KUKA KRL program: MyProgram_081().src

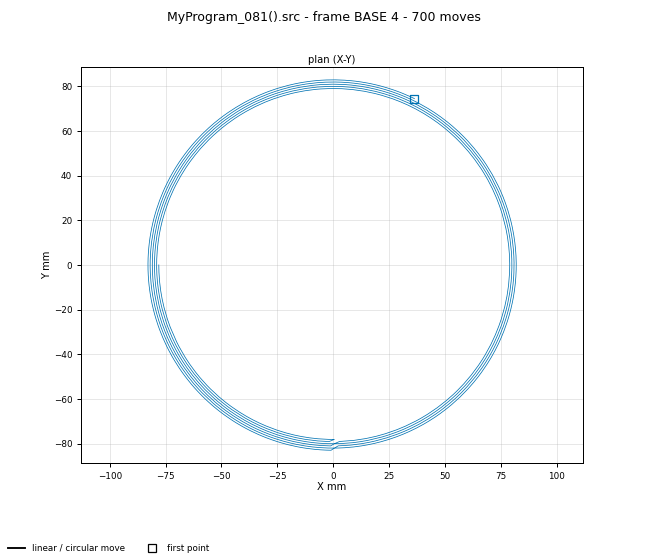
[picture p0: tool path of MyProgram_081().src in frame BASE 4, 700 of 700 moves have a stored position in this frame; points joined in program order, loops and branches not executed]
&ACCESS RVP
&REL 1
&PARAM TEMPLATE = C:\KRC\Roboter\Template\vorgabe
&PARAM EDITMASK = *
DEF MyProgram_081()
; ---- Setting reference (Base) ----
$BASE = BASE_DATA[4]

; --------------------------
; ---- Setting tool (TCP) ----
$TOOL = TOOL_DATA[3]
; --------------------------

$VEL.CP = VEL_APROX_PRINT
Startdeposition()
$VEL.CP = VEL_PRINT
LIN {X 36.3666,Y 74.5111,Z 82,A 58.7177,B 24.8945,C -2.3712,E1 25.0694,E2 385.953} C_DIS
LIN {X 34.2905,Y 75.4877,Z 82,A 60.1854,B 24.8947,C -2.3694,E1 25.0657,E2 384.4932} C_DIS
LIN {X 32.4557,Y 76.2947,Z 82,A 61.5848,B 24.8945,C -2.3714,E1 25.0621,E2 383.0926} C_DIS
LIN {X 30.7867,Y 76.9845,Z 82,A 62.9666,B 24.894,C -2.3768,E1 25.0585,E2 381.7013} C_DIS
LIN {X 28.8882,Y 77.7168,Z 82,A 64.37,B 24.8939,C -2.378,E1 25.0549,E2 380.298} C_DIS
LIN {X 26.9089,Y 78.4237,Z 82,A 65.9427,B 24.8934,C -2.3829,E1 25.0507,E2 378.7167} C_DIS
LIN {X 24.0041,Y 79.361,Z 82,A 67.8847,B 24.8938,C -2.3794,E1 25.0456,E2 376.7865} C_DIS
LIN {X 22.1137,Y 79.9088,Z 82,A 69.2831,B 24.8936,C -2.3815,E1 25.0418,E2 375.3855} C_DIS
LIN {X 19.68,Y 80.5411,Z 82,A 71.0984,B 24.8933,C -2.3849,E1 25.0369,E2 373.5648} C_DIS
LIN {X 17.1067,Y 81.1279,Z 82,A 72.799,B 24.8935,C -2.3821,E1 25.0322,E2 371.8732} C_DIS
LIN {X 15.1105,Y 81.5232,Z 82,A 74.2055,B 24.8935,C -2.3827,E1 25.0284,E2 370.4669} C_DIS
LIN {X 12.5489,Y 81.9555,Z 82,A 76.1064,B 24.8931,C -2.3864,E1 25.0231,E2 368.559} C_DIS
LIN {X 10.083,Y 82.2964,Z 82,A 77.7189,B 24.8934,C -2.3835,E1 25.0187,E2 366.9546} C_DIS
LIN {X 8.1268,Y 82.5129,Z 82,A 79.2702,B 24.8929,C -2.3894,E1 25.0143,E2 365.3903} C_DIS
LIN {X 5.0842,Y 82.7562,Z 82,A 81.2283,B 24.8933,C -2.385,E1 25.0089,E2 363.4437} C_DIS
LIN {X 2.8241,Y 82.863,Z 82,A 82.6559,B 24.8936,C -2.3809,E1 25.005,E2 362.0264} C_DIS
LIN {X 0.9507,Y 82.9063,Z 82,A 84.0039,B 24.8936,C -2.3823,E1 25.0012,E2 360.6753} C_DIS
LIN {X -1.0175,Y 82.9059,Z 82,A 85.4483,B 24.8933,C -2.3844,E1 24.9971,E2 359.2256} C_DIS
LIN {X -3.0518,Y 82.856,Z 82,A 86.8554,B 24.8933,C -2.3841,E1 24.9932,E2 357.8193} C_DIS
LIN {X -5.5817,Y 82.7225,Z 82,A 88.7172,B 24.8931,C -2.3867,E1 24.988,E2 355.9506} C_DIS
LIN {X -8.1268,Y 82.5129,Z 82,A 90.3341,B 24.8936,C -2.3815,E1 24.9835,E2 354.3454} C_DIS
LIN {X -10.1493,Y 82.2886,Z 82,A 91.9555,B 24.8931,C -2.3869,E1 24.979,E2 352.7098} C_DIS
LIN {X -13.2371,Y 81.8483,Z 82,A 93.8578,B 24.8939,C -2.3782,E1 24.9738,E2 350.8268} C_DIS
LIN {X -15.2418,Y 81.4988,Z 82,A 95.3126,B 24.8939,C -2.3785,E1 24.9698,E2 349.3697} C_DIS
LIN {X -17.2373,Y 81.1002,Z 82,A 96.8676,B 24.8936,C -2.3816,E1 24.9655,E2 347.8054} C_DIS
LIN {X -20.146,Y 80.4274,Z 82,A 98.8262,B 24.894,C -2.3767,E1 24.9602,E2 345.8559} C_DIS
LIN {X -22.2027,Y 79.8836,Z 82,A 100.1992,B 24.8944,C -2.3724,E1 24.9566,E2 344.4909} C_DIS
LIN {X -24.1319,Y 79.3222,Z 82,A 101.6507,B 24.8944,C -2.3727,E1 24.9527,E2 343.0363} C_DIS
LIN {X -26.008,Y 78.7274,Z 82,A 103.1904,B 24.894,C -2.3762,E1 24.9485,E2 341.4855} C_DIS
LIN {X -28.8882,Y 77.7168,Z 82,A 105.1706,B 24.8946,C -2.3699,E1 24.9434,E2 339.5164} C_DIS
LIN {X -30.7867,Y 76.9845,Z 82,A 106.7223,B 24.8944,C -2.3721,E1 24.9393,E2 337.956} C_DIS
LIN {X -33.5994,Y 75.7991,Z 82,A 108.8877,B 24.8945,C -2.3706,E1 24.9338,E2 335.789} C_DIS
LIN {X -36.4697,Y 74.46,Z 82,A 110.7784,B 24.8956,C -2.3589,E1 24.9291,E2 333.9215} C_DIS
LIN {X -38.1843,Y 73.5961,Z 82,A 112.225,B 24.8955,C -2.3601,E1 24.9254,E2 332.4682} C_DIS
LIN {X -40.0714,Y 72.5853,Z 82,A 113.6009,B 24.896,C -2.3547,E1 24.9221,E2 331.1012} C_DIS
LIN {X -41.9287,Y 71.5279,Z 82,A 115.0677,B 24.8962,C -2.3518,E1 24.9185,E2 329.6368} C_DIS
LIN {X -43.5515,Y 70.5523,Z 82,A 116.4661,B 24.8962,C -2.3519,E1 24.9152,E2 328.2338} C_DIS
LIN {X -45.2141,Y 69.499,Z 82,A 117.8318,B 24.8964,C -2.3495,E1 24.912,E2 326.8695} C_DIS
LIN {X -46.9061,Y 68.3685,Z 82,A 119.2443,B 24.8966,C -2.3469,E1 24.9087,E2 325.4584} C_DIS
LIN {X -49.0864,Y 66.8185,Z 82,A 121.2055,B 24.8966,C -2.3463,E1 24.9043,E2 323.4917} C_DIS
LIN {X -51.0626,Y 65.3221,Z 82,A 122.9521,B 24.8969,C -2.3437,E1 24.9004,E2 321.7452} C_DIS
LIN {X -53.3815,Y 63.4417,Z 82,A 125.1052,B 24.8971,C -2.3416,E1 24.8958,E2 319.5887} C_DIS
LIN {X -55.7296,Y 61.3887,Z 82,A 127.114,B 24.8979,C -2.3327,E1 24.8916,E2 317.5931} C_DIS
LIN {X -57.1713,Y 60.0489,Z 82,A 128.4698,B 24.8982,C -2.3294,E1 24.8889,E2 316.2396} C_DIS
LIN {X -58.6278,Y 58.6278,Z 82,A 129.8425,B 24.8986,C -2.3252,E1 24.8862,E2 314.8713} C_DIS
LIN {X -60.2074,Y 57.0028,Z 82,A 131.3189,B 24.8991,C -2.319,E1 24.8833,E2 313.4034} C_DIS
LIN {X -61.4339,Y 55.6804,Z 82,A 132.7293,B 24.899,C -2.3203,E1 24.8806,E2 311.9836} C_DIS
LIN {X -62.8251,Y 54.1052,Z 82,A 134.131,B 24.8994,C -2.3153,E1 24.8781,E2 310.5876} C_DIS
LIN {X -64.5211,Y 52.0695,Z 82,A 136.027,B 24.8997,C -2.3123,E1 24.8747,E2 308.6898} C_DIS
LIN {X -66.2877,Y 49.8008,Z 82,A 138.1202,B 24.8999,C -2.3099,E1 24.8711,E2 306.5924} C_DIS
LIN {X -67.7877,Y 47.7415,Z 82,A 139.7835,B 24.9005,C -2.3025,E1 24.8685,E2 304.9386} C_DIS
LIN {X -68.939,Y 46.0635,Z 82,A 141.1579,B 24.9009,C -2.2978,E1 24.8663,E2 303.5686} C_DIS
LIN {X -70.084,Y 44.3012,Z 82,A 142.6197,B 24.9013,C -2.294,E1 24.8641,E2 302.1085} C_DIS
LIN {X -71.1501,Y 42.5679,Z 82,A 143.9912,B 24.9017,C -2.2891,E1 24.8621,E2 300.7417} C_DIS
LIN {X -72.1734,Y 40.809,Z 82,A 145.4498,B 24.9019,C -2.2865,E1 24.8601,E2 299.2817} C_DIS
LIN {X -73.2059,Y 38.9252,Z 82,A 146.8267,B 24.9025,C -2.2793,E1 24.8583,E2 297.9146} C_DIS
LIN {X -74.2664,Y 36.8601,Z 82,A 148.6842,B 24.9024,C -2.2814,E1 24.8559,E2 296.0422} C_DIS
LIN {X -75.3811,Y 34.5271,Z 82,A 150.3979,B 24.903,C -2.2741,E1 24.8539,E2 294.3366} C_DIS
LIN {X -76.2317,Y 32.6052,Z 82,A 151.7761,B 24.9035,C -2.2678,E1 24.8524,E2 292.9658} C_DIS
LIN {X -77.0089,Y 30.7246,Z 82,A 153.2354,B 24.9038,C -2.2649,E1 24.8509,E2 291.5052} C_DIS
LIN {X -77.7168,Y 28.8882,Z 82,A 154.6452,B 24.904,C -2.2621,E1 24.8495,E2 290.0942} C_DIS
LIN {X -78.4237,Y 26.9089,Z 82,A 156.0236,B 24.9045,C -2.2557,E1 24.8482,E2 288.7233} C_DIS
LIN {X -79.0407,Y 25.04,Z 82,A 157.4772,B 24.9047,C -2.254,E1 24.8469,E2 287.2655} C_DIS
LIN {X -79.6314,Y 23.0927,Z 82,A 158.8526,B 24.9051,C -2.2488,E1 24.8459,E2 285.8945} C_DIS
LIN {X -80.1907,Y 21.0668,Z 82,A 160.3148,B 24.9055,C -2.2445,E1 24.8448,E2 284.4341} C_DIS
LIN {X -80.7558,Y 18.7798,Z 82,A 162.1107,B 24.9055,C -2.2439,E1 24.8436,E2 282.6291} C_DIS
LIN {X -81.319,Y 16.1754,Z 82,A 163.8495,B 24.9063,C -2.2353,E1 24.8427,E2 280.9006} C_DIS
LIN {X -81.6915,Y 14.1748,Z 82,A 165.3159,B 24.9065,C -2.2324,E1 24.8419,E2 279.4323} C_DIS
LIN {X -82.0148,Y 12.1657,Z 82,A 166.6819,B 24.907,C -2.2269,E1 24.8414,E2 278.0714} C_DIS
LIN {X -82.2964,Y 10.083,Z 82,A 168.1039,B 24.9074,C -2.2215,E1 24.8409,E2 276.6539} C_DIS
LIN {X -82.5566,Y 7.6534,Z 82,A 169.9271,B 24.9076,C -2.2197,E1 24.8403,E2 274.824} C_DIS
LIN {X -82.7562,Y 5.0842,Z 82,A 171.6388,B 24.9082,C -2.2121,E1 24.84,E2 273.1199} C_DIS
LIN {X -82.856,Y 3.0518,Z 82,A 173.0551,B 24.9086,C -2.2079,E1 24.8399,E2 271.7052} C_DIS
LIN {X -82.9089,Y 0.6054,Z 82,A 174.8775,B 24.9087,C -2.2061,E1 24.8398,E2 269.8763} C_DIS
LIN {X -82.8848,Y -2.1118,Z 82,A 176.5585,B 24.9096,C -2.1948,E1 24.8398,E2 268.212} C_DIS
LIN {X -82.7859,Y -4.5468,Z 82,A 178.4258,B 24.9096,C -2.1944,E1 24.8401,E2 266.3345} C_DIS
LIN {X -82.6003,Y -7.1801,Z 82,A -179.9016,B 24.9105,C -2.1846,E1 24.8405,E2 264.6752} C_DIS
LIN {X -82.407,Y -9.1388,Z 82,A -178.4886,B 24.9107,C -2.1817,E1 24.8409,E2 263.2607} C_DIS
LIN {X -82.1485,Y -11.2245,Z 82,A -177.0693,B 24.9112,C -2.1763,E1 24.8414,E2 261.8458} C_DIS
LIN {X -81.8483,Y -13.2371,Z 82,A -175.6493,B 24.9115,C -2.1723,E1 24.842,E2 260.427} C_DIS
LIN {X -81.4988,Y -15.2418,Z 82,A -174.1937,B 24.9117,C -2.1692,E1 24.8427,E2 258.97} C_DIS
LIN {X -81.1002,Y -17.2373,Z 82,A -172.616,B 24.9117,C -2.1695,E1 24.8436,E2 257.3823} C_DIS
LIN {X -80.4274,Y -20.146,Z 82,A -170.6601,B 24.9125,C -2.1603,E1 24.8449,E2 255.4368} C_DIS
LIN {X -79.8906,Y -22.178,Z 82,A -169.2822,B 24.913,C -2.154,E1 24.8459,E2 254.0661} C_DIS
LIN {X -79.3222,Y -24.1319,Z 82,A -167.7349,B 24.913,C -2.1536,E1 24.8471,E2 252.5109} C_DIS
LIN {X -78.4024,Y -26.9722,Z 82,A -165.7053,B 24.9136,C -2.1466,E1 24.8489,E2 250.4864} C_DIS
LIN {X -77.7168,Y -28.8882,Z 82,A -164.29,B 24.9139,C -2.1427,E1 24.8503,E2 249.0723} C_DIS
LIN {X -76.9209,Y -30.9428,Z 82,A -162.8596,B 24.9144,C -2.1358,E1 24.8517,E2 247.6503} C_DIS
LIN {X -76.2057,Y -32.6667,Z 82,A -161.5,B 24.9146,C -2.134,E1 24.8532,E2 246.2874} C_DIS
LIN {X -75.3529,Y -34.5876,Z 82,A -160.0387,B 24.9149,C -2.1302,E1 24.8549,E2 244.8273} C_DIS
LIN {X -74.5111,Y -36.3666,Z 82,A -158.6427,B 24.9151,C -2.1274,E1 24.8566,E2 243.4304} C_DIS
LIN {X -73.5149,Y -38.3385,Z 82,A -157.0559,B 24.9153,C -2.1249,E1 24.8586,E2 241.8412} C_DIS
LIN {X -72.1408,Y -40.8673,Z 82,A -155.0928,B 24.9158,C -2.1188,E1 24.8613,E2 239.8822} C_DIS
LIN {X -71.0815,Y -42.6824,Z 82,A -153.716,B 24.9163,C -2.113,E1 24.8632,E2 238.5123} C_DIS
LIN {X -70.0126,Y -44.414,Z 82,A -152.3013,B 24.9165,C -2.1095,E1 24.8653,E2 237.0985} C_DIS
LIN {X -68.939,Y -46.0635,Z 82,A -150.8498,B 24.9166,C -2.1086,E1 24.8675,E2 235.6419} C_DIS
LIN {X -67.7877,Y -47.7415,Z 82,A -149.4764,B 24.917,C -2.1042,E1 24.8697,E2 234.2723} C_DIS
LIN {X -66.5556,Y -49.4441,Z 82,A -148.0161,B 24.9172,C -2.1009,E1 24.8721,E2 232.8128} C_DIS
LIN {X -65.0276,Y -51.4352,Z 82,A -146.1371,B 24.9172,C -2.1008,E1 24.8754,E2 230.9252} C_DIS
LIN {X -63.4417,Y -53.3815,Z 82,A -144.4879,B 24.9177,C -2.0944,E1 24.8783,E2 229.2837} C_DIS
LIN {X -62.1125,Y -54.9223,Z 82,A -143.1152,B 24.9181,C -2.0903,E1 24.8808,E2 227.9145} C_DIS
LIN {X -60.7002,Y -56.4787,Z 82,A -141.6555,B 24.9183,C -2.0873,E1 24.8836,E2 226.4555} C_DIS
LIN {X -58.6278,Y -58.6278,Z 82,A -139.5827,B 24.9186,C -2.0832,E1 24.8876,E2 224.3836} C_DIS
LIN {X -57.1713,Y -60.0489,Z 82,A -138.1295,B 24.9187,C -2.0816,E1 24.8906,E2 222.9281} C_DIS
LIN {X -55.6307,Y -61.4784,Z 82,A -136.534,B 24.9187,C -2.0828,E1 24.8939,E2 221.3234} C_DIS
LIN {X -53.3815,Y -63.4417,Z 82,A -134.6393,B 24.9193,C -2.0741,E1 24.8978,E2 219.442} C_DIS
LIN {X -51.8085,Y -64.7326,Z 82,A -133.2273,B 24.9195,C -2.0717,E1 24.9009,E2 218.0305} C_DIS
LIN {X -50.2042,Y -65.9846,Z 82,A -131.7749,B 24.9196,C -2.0705,E1 24.9041,E2 216.5756} C_DIS
LIN {X -48.5154,Y -67.2355,Z 82,A -130.3885,B 24.9199,C -2.0662,E1 24.9072,E2 215.1946} C_DIS
LIN {X -46.8508,Y -68.4059,Z 82,A -128.9463,B 24.92,C -2.0649,E1 24.9106,E2 213.7505} C_DIS
LIN {X -45.2141,Y -69.499,Z 82,A -127.5411,B 24.9201,C -2.0641,E1 24.9138,E2 212.3427} C_DIS
LIN {X -43.4949,Y -70.5877,Z 82,A -125.9412,B 24.9198,C -2.0675,E1 24.9177,E2 210.7296} C_DIS
LIN {X -40.8673,Y -72.1408,Z 82,A -124.0142,B 24.9205,C -2.0593,E1 24.9223,E2 208.8163} C_DIS
LIN {X -39.0255,Y -73.1531,Z 82,A -122.5977,B 24.9207,C -2.0564,E1 24.9258,E2 207.4028} C_DIS
LIN {X -37.1946,Y -74.1006,Z 82,A -121.2297,B 24.921,C -2.053,E1 24.9292,E2 206.0392} C_DIS
LIN {X -35.2165,Y -75.0602,Z 82,A -119.7594,B 24.9212,C -2.0498,E1 24.9329,E2 204.5727} C_DIS
LIN {X -33.5383,Y -75.8258,Z 82,A -118.4118,B 24.9212,C -2.0505,E1 24.9363,E2 203.2202} C_DIS
LIN {X -31.7291,Y -76.6009,Z 82,A -117.005,B 24.9212,C -2.0505,E1 24.9399,E2 201.8103} C_DIS
LIN {X -29.7773,Y -77.3801,Z 82,A -115.4333,B 24.921,C -2.0526,E1 24.944,E2 200.2302} C_DIS
LIN {X -27.646,Y -78.1659,Z 82,A -113.836,B 24.921,C -2.052,E1 24.9482,E2 198.6309} C_DIS
LIN {X -25.04,Y -79.0407,Z 82,A -112.0332,B 24.9214,C -2.0477,E1 24.953,E2 196.8352} C_DIS
LIN {X -22.7292,Y -79.7344,Z 82,A -110.2445,B 24.9212,C -2.0502,E1 24.9578,E2 195.0376} C_DIS
LIN {X -20.0812,Y -80.4432,Z 82,A -108.55,B 24.9217,C -2.0432,E1 24.9624,E2 193.3573} C_DIS
LIN {X -18.1662,Y -80.8976,Z 82,A -107.1456,B 24.9217,C -2.0438,E1 24.9662,E2 191.9496} C_DIS
LIN {X -16.1754,Y -81.319,Z 82,A -105.6975,B 24.9217,C -2.0445,E1 24.9702,E2 190.4982} C_DIS
LIN {X -14.1748,Y -81.6915,Z 82,A -104.2905,B 24.9217,C -2.044,E1 24.974,E2 189.0908} C_DIS
LIN {X -12.1657,Y -82.0148,Z 82,A -102.8832,B 24.9217,C -2.0437,E1 24.9779,E2 187.6831} C_DIS
LIN {X -10.083,Y -82.2964,Z 82,A -101.4707,B 24.9217,C -2.0422,E1 24.9818,E2 186.273} C_DIS
LIN {X -8.1268,Y -82.5129,Z 82,A -100.0699,B 24.9217,C -2.0433,E1 24.9857,E2 184.8688} C_DIS
LIN {X -5.6119,Y -82.7205,Z 82,A -98.2133,B 24.9214,C -2.0467,E1 24.9909,E2 183.0034} C_DIS
LIN {X -3.0518,Y -82.856,Z 82,A -96.5545,B 24.9217,C -2.0434,E1 24.9955,E2 181.3519} C_DIS
LIN {X -0.9507,Y -82.9063,Z 82,A -95.1862,B 24.9219,C -2.0412,E1 24.9993,E2 179.9891} C_DIS
LIN {X -0.9507,Y -82.9063,Z 82,A -95.1862,B 24.9219,C -2.0412,E1 24.9993,E2 179.9891} C_DIS
Enddeposition()
LIN {X 0.5436,Y -81.9382,Z 82,A -94.7456,B 24.9219,C -2.0405,E1 25.0006,E2 179.55} C_DIS
Startdeposition()
$VEL.CP = VEL_PRINT
LIN {X -2.3454,Y -81.9084,Z 82,A -97.1195,B 24.9228,C -2.0297,E1 24.9939,E2 181.9498} C_DIS
LIN {X -6.226,Y -81.7055,Z 82,A -99.7202,B 24.9225,C -2.033,E1 24.9866,E2 184.5435} C_DIS
LIN {X -9.2508,Y -81.4184,Z 82,A -101.8577,B 24.9225,C -2.0328,E1 24.9807,E2 186.6827} C_DIS
LIN {X -12.664,Y -80.9574,Z 82,A -104.2918,B 24.9225,C -2.0326,E1 24.974,E2 189.1192} C_DIS
LIN {X -16.2227,Y -80.3203,Z 82,A -106.7628,B 24.9223,C -2.0352,E1 24.9672,E2 191.5867} C_DIS
LIN {X -19.0809,Y -79.69,Z 82,A -108.8501,B 24.9223,C -2.035,E1 24.9615,E2 193.6772} C_DIS
LIN {X -22.2862,Y -78.8529,Z 82,A -111.0933,B 24.9221,C -2.0386,E1 24.9555,E2 195.9154} C_DIS
LIN {X -26.2246,Y -77.632,Z 82,A -113.6473,B 24.9212,C -2.0501,E1 24.9487,E2 198.4464} C_DIS
LIN {X -28.3647,Y -76.8764,Z 82,A -115.416,B 24.9215,C -2.0463,E1 24.944,E2 200.2278} C_DIS
LIN {X -30.7313,Y -75.961,Z 82,A -117.4251,B 24.9219,C -2.0413,E1 24.9388,E2 202.2531} C_DIS
LIN {X -33.8409,Y -74.6276,Z 82,A -119.8587,B 24.9219,C -2.042,E1 24.9326,E2 204.6909} C_DIS
LIN {X -36.3834,Y -73.4214,Z 82,A -121.6585,B 24.9213,C -2.049,E1 24.9281,E2 206.4787} C_DIS
LIN {X -38.8459,Y -72.1492,Z 82,A -123.6739,B 24.9213,C -2.0493,E1 24.9231,E2 208.4988} C_DIS
LIN {X -41.3243,Y -70.7597,Z 82,A -125.772,B 24.9213,C -2.049,E1 24.918,E2 210.604} C_DIS
LIN {X -43.6656,Y -69.3387,Z 82,A -127.6745,B 24.921,C -2.0522,E1 24.9135,E2 212.5048} C_DIS
LIN {X -46.4991,Y -67.4714,Z 82,A -130.0207,B 24.9207,C -2.0567,E1 24.908,E2 214.8481} C_DIS
LIN {X -49.2408,Y -65.4965,Z 82,A -132.3955,B 24.9204,C -2.0604,E1 24.9027,E2 217.2225} C_DIS
LIN {X -51.9306,Y -63.3864,Z 82,A -134.8712,B 24.9202,C -2.0624,E1 24.8973,E2 219.7026} C_DIS
LIN {X -53.8172,Y -61.7913,Z 82,A -136.7556,B 24.9203,C -2.0614,E1 24.8933,E2 221.5966} C_DIS
LIN {X -58.6217,Y -57.2553,Z 82,A -140.9587,B 24.9187,C -2.0822,E1 24.8849,E2 225.7678} C_DIS
LIN {X -60.3993,Y -55.3749,Z 82,A -142.9677,B 24.9188,C -2.0808,E1 24.8811,E2 227.789} C_DIS
LIN {X -62.4942,Y -52.9997,Z 82,A -145.471,B 24.919,C -2.078,E1 24.8765,E2 230.3102} C_DIS
LIN {X -64.9751,Y -49.927,Z 82,A -148.3322,B 24.9187,C -2.0819,E1 24.8715,E2 233.1756} C_DIS
LIN {X -68.0897,Y -45.5892,Z 82,A -151.6414,B 24.9171,C -2.1025,E1 24.8663,E2 236.4521} C_DIS
LIN {X -69.2197,Y -43.8557,Z 82,A -153.2472,B 24.9171,C -2.102,E1 24.8639,E2 238.0673} C_DIS
LIN {X -70.9401,Y -41.0121,Z 82,A -155.4718,B 24.9164,C -2.1107,E1 24.8607,E2 240.2825} C_DIS
LIN {X -72.3116,Y -38.5441,Z 82,A -157.3239,B 24.9158,C -2.1192,E1 24.8582,E2 242.124} C_DIS
LIN {X -73.5937,Y -36.0354,Z 82,A -159.2388,B 24.9152,C -2.1261,E1 24.8558,E2 244.0329} C_DIS
LIN {X -74.593,Y -33.9178,Z 82,A -161.1658,B 24.9155,C -2.1231,E1 24.8536,E2 245.9776} C_DIS
LIN {X -75.9121,Y -30.8514,Z 82,A -163.464,B 24.9149,C -2.1307,E1 24.8511,E2 248.2704} C_DIS
LIN {X -77.0814,Y -27.8028,Z 82,A -165.8401,B 24.9145,C -2.1349,E1 24.8488,E2 250.6498} C_DIS
LIN {X -78.1488,Y -24.6449,Z 82,A -168.1952,B 24.914,C -2.1411,E1 24.8467,E2 253.0035} C_DIS
LIN {X -79.0854,Y -21.4468,Z 82,A -170.5128,B 24.9134,C -2.1485,E1 24.845,E2 255.317} C_DIS
LIN {X -79.8523,Y -18.3866,Z 82,A -173.0081,B 24.9134,C -2.1477,E1 24.8434,E2 257.8287} C_DIS
LIN {X -80.7667,Y -13.831,Z 82,A -175.7493,B 24.9116,C -2.1709,E1 24.842,E2 260.5309} C_DIS
LIN {X -81.1564,Y -11.3196,Z 82,A -177.7691,B 24.9116,C -2.1701,E1 24.8411,E2 262.5645} C_DIS
LIN {X -81.5003,Y -8.4944,Z 82,A -179.9756,B 24.9116,C -2.1708,E1 24.8404,E2 264.7825} C_DIS
LIN {X -81.8486,Y -3.9273,Z 82,A 176.997,B 24.9104,C -2.1854,E1 24.8399,E2 267.7932} C_DIS
LIN {X -81.939,Y -0.7395,Z 82,A 174.7493,B 24.9099,C -2.1921,E1 24.8398,E2 270.0386} C_DIS
LIN {X -81.9133,Y 2.1842,Z 82,A 172.7159,B 24.9093,C -2.1989,E1 24.8398,E2 272.0681} C_DIS
LIN {X -81.7157,Y 6.0961,Z 82,A 170.1967,B 24.9081,C -2.2133,E1 24.8403,E2 274.568} C_DIS
LIN {X -81.2855,Y 10.3514,Z 82,A 166.5726,B 24.9087,C -2.2065,E1 24.8414,E2 278.23} C_DIS
LIN {X -80.3185,Y 16.2312,Z 82,A 162.3829,B 24.9076,C -2.2192,E1 24.8435,E2 282.4143} C_DIS
LIN {X -79.4539,Y 20.0417,Z 82,A 159.3218,B 24.9076,C -2.2193,E1 24.8456,E2 285.4929} C_DIS
LIN {X -78.4999,Y 23.5002,Z 82,A 156.9548,B 24.9067,C -2.2307,E1 24.8474,E2 287.8464} C_DIS
LIN {X -77.0866,Y 27.7885,Z 82,A 154.2829,B 24.9048,C -2.2529,E1 24.8498,E2 290.4806} C_DIS
LIN {X -75.8979,Y 30.8862,Z 82,A 151.9577,B 24.9042,C -2.2598,E1 24.8522,E2 292.8022} C_DIS
LIN {X -74.6875,Y 33.708,Z 82,A 149.484,B 24.9044,C -2.2578,E1 24.855,E2 295.2943} C_DIS
LIN {X -73.2997,Y 36.6289,Z 82,A 147.0715,B 24.9041,C -2.2606,E1 24.858,E2 297.7132} C_DIS
LIN {X -70.6017,Y 41.5916,Z 82,A 143.5876,B 24.9021,C -2.284,E1 24.8627,E2 301.1596} C_DIS
LIN {X -69.0343,Y 44.1445,Z 82,A 141.4676,B 24.9017,C -2.2892,E1 24.8659,E2 303.2779} C_DIS
LIN {X -67.3282,Y 46.7051,Z 82,A 139.3303,B 24.9011,C -2.2955,E1 24.8692,E2 305.4109} C_DIS
LIN {X -64.8816,Y 50.0482,Z 82,A 135.3725,B 24.9028,C -2.2756,E1 24.876,E2 309.4348} C_DIS
LIN {X -61.9823,Y 53.5986,Z 82,A 133.3815,B 24.8994,C -2.3155,E1 24.8795,E2 311.34} C_DIS
LIN {X -60.3528,Y 55.4256,Z 82,A 131.2213,B 24.9001,C -2.3079,E1 24.8835,E2 313.5278} C_DIS
LIN {X -58.1831,Y 57.6993,Z 82,A 129.2686,B 24.899,C -2.3197,E1 24.8873,E2 315.4608} C_DIS
LIN {X -56.048,Y 59.7753,Z 82,A 126.7867,B 24.8995,C -2.314,E1 24.8924,E2 317.9664} C_DIS
LIN {X -53.553,Y 62.0221,Z 82,A 124.686,B 24.8985,C -2.3258,E1 24.8968,E2 320.0474} C_DIS
LIN {X -50.2871,Y 64.6976,Z 82,A 122.0707,B 24.8972,C -2.3411,E1 24.9024,E2 322.6359} C_DIS
LIN {X -45.3387,Y 68.2564,Z 82,A 117.5214,B 24.8971,C -2.3419,E1 24.9128,E2 327.1989} C_DIS
LIN {X -42.7724,Y 69.8931,Z 82,A 115.3527,B 24.8968,C -2.3448,E1 24.9179,E2 329.3677} C_DIS
LIN {X -40.361,Y 71.3138,Z 82,A 112.9042,B 24.8977,C -2.3349,E1 24.9239,E2 331.8469} C_DIS
LIN {X -35.8384,Y 73.6899,Z 82,A 109.765,B 24.8962,C -2.3524,E1 24.9317,E2 334.9529} C_DIS
LIN {X -33.0723,Y 74.972,Z 82,A 107.6559,B 24.8958,C -2.3562,E1 24.937,E2 337.058} C_DIS
LIN {X -28.5189,Y 76.8191,Z 82,A 104.4745,B 24.8948,C -2.3679,E1 24.9452,E2 340.2186} C_DIS
LIN {X -26.0036,Y 77.7065,Z 82,A 102.3152,B 24.8953,C -2.362,E1 24.951,E2 342.396} C_DIS
LIN {X -22.8598,Y 78.6899,Z 82,A 99.5754,B 24.8962,C -2.3525,E1 24.9584,E2 345.1631} C_DIS
LIN {X -19.2461,Y 79.6497,Z 82,A 97.3645,B 24.8949,C -2.3662,E1 24.9643,E2 347.3446} C_DIS
LIN {X -15.9368,Y 80.3783,Z 82,A 94.3004,B 24.8965,C -2.3488,E1 24.9728,E2 350.4535} C_DIS
LIN {X -12.151,Y 81.0367,Z 82,A 92.6384,B 24.8938,C -2.3794,E1 24.9772,E2 352.0443} C_DIS
LIN {X -7.1036,Y 81.6344,Z 82,A 89.0636,B 24.8936,C -2.3808,E1 24.9871,E2 355.6181} C_DIS
LIN {X -3.4048,Y 81.8711,Z 82,A 86.1286,B 24.8944,C -2.3719,E1 24.9953,E2 358.575} C_DIS
LIN {X 0.9377,Y 81.9369,Z 82,A 83.1329,B 24.8943,C -2.3738,E1 25.0037,E2 361.5663} C_DIS
LIN {X 3.8857,Y 81.8504,Z 82,A 81.1168,B 24.8941,C -2.3752,E1 25.0093,E2 363.5784} C_DIS
LIN {X 6.7881,Y 81.6605,Z 82,A 79.1252,B 24.8941,C -2.3764,E1 25.0148,E2 365.5664} C_DIS
LIN {X 9.3512,Y 81.4066,Z 82,A 77.2108,B 24.8944,C -2.3728,E1 25.0202,E2 367.4878} C_DIS
LIN {X 12.5745,Y 80.9712,Z 82,A 75.3368,B 24.8934,C -2.3839,E1 25.0253,E2 369.3338} C_DIS
LIN {X 14.5701,Y 80.636,Z 82,A 73.686,B 24.894,C -2.3765,E1 25.0299,E2 371.0005} C_DIS
LIN {X 17.4359,Y 80.0652,Z 82,A 71.4358,B 24.8946,C -2.3695,E1 25.036,E2 373.2645} C_DIS
LIN {X 20.7245,Y 79.2784,Z 82,A 68.7841,B 24.8955,C -2.3596,E1 25.0433,E2 375.9356} C_DIS
LIN {X 23.7888,Y 78.4142,Z 82,A 66.8698,B 24.8949,C -2.3672,E1 25.0483,E2 377.8286} C_DIS
LIN {X 26.2191,Y 77.6338,Z 82,A 65.1593,B 24.8948,C -2.368,E1 25.0529,E2 379.5341} C_DIS
LIN {X 29.4248,Y 76.4776,Z 82,A 62.7168,B 24.8951,C -2.364,E1 25.0593,E2 381.9808} C_DIS
LIN {X 32.6317,Y 75.1641,Z 82,A 60.4217,B 24.8951,C -2.3653,E1 25.0651,E2 384.2675} C_DIS
LIN {X 35.565,Y 73.8213,Z 82,A 58.2234,B 24.8951,C -2.3644,E1 25.0707,E2 386.4623} C_DIS
LIN {X 38.2464,Y 72.4684,Z 82,A 56.0658,B 24.8955,C -2.3599,E1 25.0761,E2 388.6244} C_DIS
LIN {X 42.4451,Y 70.092,Z 82,A 52.0586,B 24.8976,C -2.3359,E1 25.0858,E2 392.6763} C_DIS
LIN {X 45.39,Y 68.2225,Z 82,A 50.1691,B 24.8965,C -2.3487,E1 25.0902,E2 394.5292} C_DIS
LIN {X 48.1996,Y 66.267,Z 82,A 47.8919,B 24.8965,C -2.3483,E1 25.0953,E2 396.7995} C_DIS
LIN {X 51.1536,Y 64.0153,Z 82,A 45.2221,B 24.8971,C -2.3414,E1 25.1012,E2 399.4758} C_DIS
LIN {X 53.4502,Y 62.1103,Z 82,A 42.4728,B 24.8993,C -2.3169,E1 25.1072,E2 402.2722} C_DIS
LIN {X 56.2326,Y 59.6017,Z 82,A 40.7074,B 24.8974,C -2.3381,E1 25.1106,E2 403.9804} C_DIS
LIN {X 58.2791,Y 57.6021,Z 82,A 38.6782,B 24.8979,C -2.333,E1 25.1147,E2 406.0131} C_DIS
LIN {X 60.2969,Y 55.4865,Z 82,A 36.2663,B 24.8993,C -2.317,E1 25.1193,E2 408.4522} C_DIS
LIN {X 62.9709,Y 52.4321,Z 82,A 33.7881,B 24.8989,C -2.3218,E1 25.1238,E2 410.9078} C_DIS
LIN {X 65.0497,Y 49.8302,Z 82,A 31.0454,B 24.9005,C -2.3032,E1 25.1285,E2 413.6816} C_DIS
LIN {X 67.2389,Y 46.8336,Z 82,A 28.9029,B 24.8998,C -2.3111,E1 25.132,E2 415.7951} C_DIS
LIN {X 68.5882,Y 44.8353,Z 82,A 27.0812,B 24.9005,C -2.3025,E1 25.1348,E2 417.6281} C_DIS
LIN {X 71.2115,Y 40.5399,Z 82,A 23.5949,B 24.9012,C -2.2942,E1 25.1398,E2 421.1159} C_DIS
LIN {X 74.024,Y 35.1433,Z 82,A 19.6426,B 24.9014,C -2.2922,E1 25.1448,E2 425.0519} C_DIS
LIN {X 75.0022,Y 33.0029,Z 82,A 17.9767,B 24.9019,C -2.2869,E1 25.1467,E2 426.7213} C_DIS
LIN {X 76.0619,Y 30.4834,Z 82,A 16.0839,B 24.9023,C -2.282,E1 25.1487,E2 428.6152} C_DIS
LIN {X 77.013,Y 27.9904,Z 82,A 13.8134,B 24.9039,C -2.2636,E1 25.1509,E2 430.9166} C_DIS
LIN {X 78.2412,Y 24.3471,Z 82,A 10.6004,B 24.906,C -2.2388,E1 25.1537,E2 434.1699} C_DIS
LIN {X 79.3246,Y 20.5446,Z 82,A 9.0383,B 24.9034,C -2.2692,E1 25.1548,E2 435.6513} C_DIS
LIN {X 79.7826,Y 18.6884,Z 82,A 7.3224,B 24.9048,C -2.2528,E1 25.1559,E2 437.396} C_DIS
LIN {X 80.2264,Y 16.68,Z 82,A 5.8085,B 24.9054,C -2.2459,E1 25.1568,E2 438.9173} C_DIS
LIN {X 80.8563,Y 13.2954,Z 82,A 3.458,B 24.9058,C -2.2403,E1 25.1579,E2 441.2673} C_DIS
LIN {X 81.3226,Y 10.0647,Z 82,A 1.3642,B 24.9059,C -2.2392,E1 25.1587,E2 443.3513} C_DIS
LIN {X 81.6137,Y 7.3277,Z 82,A -0.7479,B 24.907,C -2.2271,E1 25.1593,E2 445.4795} C_DIS
LIN {X 81.8432,Y 4.0461,Z 82,A -3.0103,B 24.9075,C -2.221,E1 25.1597,E2 447.7428} C_DIS
LIN {X 81.9392,Y 0.7102,Z 82,A -5.3424,B 24.9081,C -2.2136,E1 25.1597,E2 450.0785} C_DIS
LIN {X 81.9113,Y -2.2493,Z 82,A -7.3474,B 24.9085,C -2.2091,E1 25.1597,E2 452.0821} C_DIS
LIN {X 81.7681,Y -5.3358,Z 82,A -9.4601,B 24.9089,C -2.2038,E1 25.1594,E2 454.195} C_DIS
LIN {X 81.536,Y -8.1531,Z 82,A -11.5188,B 24.9096,C -2.1948,E1 25.1588,E2 456.2627} C_DIS
LIN {X 81.1364,Y -11.4603,Z 82,A -13.7029,B 24.9099,C -2.1921,E1 25.158,E2 458.4403} C_DIS
LIN {X 80.6375,Y -14.562,Z 82,A -15.6578,B 24.9098,C -2.193,E1 25.1571,E2 460.3816} C_DIS
LIN {X 80.2127,Y -16.7464,Z 82,A -17.4773,B 24.9109,C -2.1794,E1 25.1561,E2 462.2224} C_DIS
LIN {X 79.5661,Y -19.5889,Z 82,A -19.5019,B 24.9114,C -2.1735,E1 25.1548,E2 464.2494} C_DIS
LIN {X 78.7969,Y -22.4839,Z 82,A -21.6067,B 24.912,C -2.1666,E1 25.1533,E2 466.3584} C_DIS
LIN {X 77.9737,Y -25.1905,Z 82,A -23.8188,B 24.9131,C -2.1528,E1 25.1514,E2 468.5903} C_DIS
LIN {X 76.4056,Y -29.6103,Z 82,A -26.8443,B 24.9132,C -2.151,E1 25.1485,E2 471.6033} C_DIS
LIN {X 75.1882,Y -32.5764,Z 82,A -29.0232,B 24.9136,C -2.1463,E1 25.1461,E2 473.7814} C_DIS
LIN {X 73.8931,Y -35.4156,Z 82,A -31.1628,B 24.914,C -2.1411,E1 25.1436,E2 475.9216} C_DIS
LIN {X 72.5362,Y -38.1177,Z 82,A -33.2897,B 24.9146,C -2.1345,E1 25.1409,E2 478.0529} C_DIS
LIN {X 70.789,Y -41.2748,Z 82,A -35.6382,B 24.9146,C -2.1328,E1 25.1377,E2 480.3931} C_DIS
LIN {X 69.0228,Y -44.1623,Z 82,A -38.4991,B 24.9165,C -2.1102,E1 25.1334,E2 483.2928} C_DIS
LIN {X 66.3731,Y -48.0547,Z 82,A -41.2307,B 24.9158,C -2.1192,E1 25.1291,E2 485.9898} C_DIS
LIN {X 64.979,Y -49.9219,Z 82,A -43.6434,B 24.9181,C -2.0898,E1 25.1249,E2 488.4606} C_DIS
LIN {X 62.9024,Y -52.5145,Z 82,A -45.8861,B 24.9184,C -2.0863,E1 25.1209,E2 490.7013} C_DIS
LIN {X 60.2956,Y -55.4879,Z 82,A -48.5404,B 24.9186,C -2.0829,E1 25.1159,E2 493.352} C_DIS
LIN {X 56.7563,Y -59.1032,Z 82,A -51.8705,B 24.9188,C -2.0809,E1 25.1093,E2 496.6725} C_DIS
LIN {X 53.0087,Y -62.4865,Z 82,A -54.9496,B 24.9183,C -2.0872,E1 25.1029,E2 499.7246} C_DIS
LIN {X 50.5214,Y -64.5135,Z 82,A -57.4842,B 24.9194,C -2.0731,E1 25.0974,E2 502.2831} C_DIS
LIN {X 47.7384,Y -66.5994,Z 82,A -59.9397,B 24.9199,C -2.0673,E1 25.0918,E2 504.7434} C_DIS
LIN {X 45.6002,Y -68.0826,Z 82,A -61.5875,B 24.9197,C -2.0691,E1 25.088,E2 506.3815} C_DIS
LIN {X 43.0006,Y -69.7541,Z 82,A -64.1054,B 24.9209,C -2.0539,E1 25.082,E2 508.9274} C_DIS
LIN {X 40.4711,Y -71.2511,Z 82,A -65.9288,B 24.9206,C -2.0574,E1 25.0776,E2 510.737} C_DIS
LIN {X 37.2999,Y -72.96,Z 82,A -68.7813,B 24.9217,C -2.0428,E1 25.0705,E2 513.616} C_DIS
LIN {X 34.0338,Y -74.5407,Z 82,A -70.8963,B 24.921,C -2.0519,E1 25.0652,E2 515.7042} C_DIS
LIN {X 31.255,Y -75.7478,Z 82,A -73.013,B 24.9213,C -2.0489,E1 25.0598,E2 517.823} C_DIS
LIN {X 28.2983,Y -76.9007,Z 82,A -75.1246,B 24.9213,C -2.0492,E1 25.0543,E2 519.9292} C_DIS
LIN {X 24.8913,Y -78.0705,Z 82,A -77.5051,B 24.9212,C -2.0503,E1 25.048,E2 522.3025} C_DIS
LIN {X 21.4699,Y -79.0791,Z 82,A -80.126,B 24.9217,C -2.0437,E1 25.0409,E2 524.9347} C_DIS
LIN {X 18.6272,Y -79.7967,Z 82,A -82.1772,B 24.9218,C -2.0417,E1 25.0354,E2 526.9877} C_DIS
LIN {X 15.6886,Y -80.4261,Z 82,A -84.4171,B 24.9223,C -2.0356,E1 25.0292,E2 529.239} C_DIS
LIN {X 12.5548,Y -80.9743,Z 82,A -86.5376,B 24.9222,C -2.0371,E1 25.0234,E2 531.3539} C_DIS
LIN {X 9.091,Y -81.4371,Z 82,A -88.7831,B 24.9218,C -2.0415,E1 25.0172,E2 533.5872} C_DIS
LIN {X 5.1633,Y -81.7796,Z 82,A -91.6961,B 24.9223,C -2.0355,E1 25.009,E2 536.513} C_DIS
LIN {X 2.5399,Y -81.9024,Z 82,A -93.5637,B 24.9224,C -2.0339,E1 25.0038,E2 538.3838} C_DIS
LIN {X 0.5436,Y -81.9382,Z 82,A -94.7445,B 24.922,C -2.04,E1 25.0006,E2 539.55} C_DIS
Enddeposition()
LIN {X 0.5436,Y -81.9382,Z 82,A -94.7445,B 24.922,C -2.04,E1 25.0006,E2 539.55} C_DIS
Startdeposition()
$VEL.CP = VEL_PRINT
LIN {X 2.2707,Y -80.9413,Z 82,A -92.7754,B 24.9189,C -2.0794,E1 25.0063,E2 537.4878} C_DIS
LIN {X 7.8512,Y -80.5924,Z 82,A -88.8925,B 24.9189,C -2.079,E1 25.0171,E2 533.6077} C_DIS
LIN {X 12.8632,Y -79.9462,Z 82,A -85.1693,B 24.9184,C -2.0858,E1 25.0275,E2 529.8716} C_DIS
LIN {X 15.9664,Y -79.3838,Z 82,A -83.0036,B 24.9184,C -2.0856,E1 25.0334,E2 527.7088} C_DIS
LIN {X 18.7413,Y -78.7756,Z 82,A -81.0084,B 24.9184,C -2.087,E1 25.0388,E2 525.713} C_DIS
LIN {X 23.8773,Y -77.3725,Z 82,A -77.4751,B 24.9186,C -2.084,E1 25.0483,E2 522.1929} C_DIS
LIN {X 28.6549,Y -75.7331,Z 82,A -73.6844,B 24.9177,C -2.0951,E1 25.0583,E2 518.3833} C_DIS
LIN {X 31.6653,Y -74.525,Z 82,A -71.4374,B 24.9175,C -2.0969,E1 25.0641,E2 516.1373} C_DIS
LIN {X 33.8987,Y -73.5362,Z 82,A -68.6473,B 24.9147,C -2.1329,E1 25.0714,E2 513.269} C_DIS
LIN {X 38.1089,Y -71.4458,Z 82,A -66.5574,B 24.9173,C -2.0995,E1 25.0763,E2 511.2641} C_DIS
LIN {X 42.5064,Y -68.9205,Z 82,A -62.7745,B 24.9163,C -2.1121,E1 25.0855,E2 507.4629} C_DIS
LIN {X 45.8946,Y -66.7117,Z 82,A -60.1905,B 24.9166,C -2.1089,E1 25.0915,E2 504.8951} C_DIS
LIN {X 48.1876,Y -65.075,Z 82,A -57.4941,B 24.9145,C -2.1353,E1 25.0977,E2 502.1457} C_DIS
LIN {X 52.2646,Y -61.8476,Z 82,A -54.3291,B 24.9152,C -2.127,E1 25.1045,E2 499.0125} C_DIS
LIN {X 54.7982,Y -59.6136,Z 82,A -51.8568,B 24.9145,C -2.1351,E1 25.1096,E2 496.5309} C_DIS
LIN {X 57.3483,Y -57.1653,Z 82,A -49.2873,B 24.9138,C -2.1433,E1 25.1147,E2 493.9528} C_DIS
LIN {X 59.9301,Y -54.4532,Z 82,A -46.6714,B 24.9134,C -2.1488,E1 25.1197,E2 491.3353} C_DIS
LIN {X 63.9734,Y -49.6396,Z 82,A -42.3605,B 24.9128,C -2.1559,E1 25.1274,E2 487.0275} C_DIS
LIN {X 66.6158,Y -46.0325,Z 82,A -39.7374,B 24.9135,C -2.1471,E1 25.1316,E2 484.438} C_DIS
LIN {X 68.1816,Y -43.6793,Z 82,A -36.9191,B 24.9109,C -2.1791,E1 25.136,E2 481.5581} C_DIS
LIN {X 69.6646,Y -41.2729,Z 82,A -34.6104,B 24.9096,C -2.1949,E1 25.1393,E2 479.224} C_DIS
LIN {X 71.409,Y -38.1785,Z 82,A -32.659,B 24.9105,C -2.1838,E1 25.1419,E2 477.309} C_DIS
LIN {X 72.8345,Y -35.3817,Z 82,A -30.5155,B 24.9102,C -2.1879,E1 25.1445,E2 475.1674} C_DIS
LIN {X 74.2236,Y -32.3644,Z 82,A -28.3506,B 24.9102,C -2.1889,E1 25.147,E2 473.0118} C_DIS
LIN {X 76.1925,Y -27.4123,Z 82,A -24.7693,B 24.9097,C -2.1942,E1 25.1506,E2 469.438} C_DIS
LIN {X 77.6212,Y -23.0555,Z 82,A -21.2201,B 24.908,C -2.2141,E1 25.1537,E2 465.8617} C_DIS
LIN {X 78.4564,Y -20.0304,Z 82,A -19.1311,B 24.9078,C -2.2168,E1 25.1552,E2 463.7784} C_DIS
LIN {X 79.0985,Y -17.3215,Z 82,A -17.1465,B 24.9073,C -2.2235,E1 25.1564,E2 461.7895} C_DIS
LIN {X 79.9787,Y -12.6529,Z 82,A -13.934,B 24.9068,C -2.2293,E1 25.158,E2 458.5822} C_DIS
LIN {X 80.5124,Y -8.6255,Z 82,A -10.9071,B 24.9056,C -2.2434,E1 25.159,E2 455.5399} C_DIS
LIN {X 80.78,Y -5.5874,Z 82,A -8.7815,B 24.9051,C -2.2493,E1 25.1595,E2 453.413} C_DIS
LIN {X 80.897,Y -3.5055,Z 82,A -7.0137,B 24.9039,C -2.2635,E1 25.1597,E2 451.622} C_DIS
LIN {X 80.9674,Y 1.0463,Z 82,A -3.9871,B 24.9035,C -2.2674,E1 25.1597,E2 448.6043} C_DIS
LIN {X 80.8776,Y 3.9573,Z 82,A -1.9074,B 24.9029,C -2.2746,E1 25.1595,E2 446.52} C_DIS
LIN {X 80.6705,Y 7.0033,Z 82,A 0.2203,B 24.9024,C -2.2803,E1 25.159,E2 444.3914} C_DIS
LIN {X 80.2324,Y 10.9353,Z 82,A 2.9951,B 24.9018,C -2.2883,E1 25.1581,E2 441.6142} C_DIS
LIN {X 79.7707,Y 13.908,Z 82,A 5.11,B 24.9012,C -2.2945,E1 25.1571,E2 439.497} C_DIS
LIN {X 79.3179,Y 16.2874,Z 82,A 7.166,B 24.8998,C -2.311,E1 25.1559,E2 437.4141} C_DIS
LIN {X 78.4585,Y 20.0225,Z 82,A 9.538,B 24.9,C -2.3081,E1 25.1543,E2 435.0626} C_DIS
LIN {X 77.1297,Y 24.6517,Z 82,A 12.7833,B 24.8996,C -2.313,E1 25.1518,E2 431.8242} C_DIS
LIN {X 75.9834,Y 27.9858,Z 82,A 15.2458,B 24.8991,C -2.3193,E1 25.1495,E2 429.3607} C_DIS
LIN {X 74.8778,Y 30.8225,Z 82,A 17.441,B 24.8984,C -2.3268,E1 25.1472,E2 427.1599} C_DIS
LIN {X 73.9972,Y 32.8815,Z 82,A 19.0858,B 24.8979,C -2.3332,E1 25.1453,E2 425.5089} C_DIS
LIN {X 71.0903,Y 38.7661,Z 82,A 23.6051,B 24.8971,C -2.3419,E1 25.1396,E2 420.9931} C_DIS
LIN {X 68.4859,Y 43.202,Z 82,A 27.2458,B 24.8962,C -2.3515,E1 25.1344,E2 417.3484} C_DIS
LIN {X 66.8228,Y 45.7327,Z 82,A 29.1448,B 24.8965,C -2.3491,E1 25.1314,E2 415.4643} C_DIS
LIN {X 65.5248,Y 47.5733,Z 82,A 31.3755,B 24.8943,C -2.3734,E1 25.1277,E2 413.1871} C_DIS
LIN {X 61.8295,Y 52.2858,Z 82,A 36.299,B 24.8914,C -2.4052,E1 25.1189,E2 408.2111} C_DIS
LIN {X 58.4702,Y 56.017,Z 82,A 38.733,B 24.8939,C -2.3774,E1 25.1144,E2 405.8535} C_DIS
LIN {X 55.9859,Y 58.5002,Z 82,A 41.5694,B 24.8925,C -2.3936,E1 25.1086,E2 402.9906} C_DIS
LIN {X 51.9494,Y 62.1121,Z 82,A 44.9982,B 24.893,C -2.3883,E1 25.1015,E2 399.5877} C_DIS
LIN {X 48.4672,Y 64.8659,Z 82,A 48.1847,B 24.8923,C -2.3954,E1 25.0944,E2 396.3963} C_DIS
LIN {X 45.9079,Y 66.7024,Z 82,A 50.321,B 24.8923,C -2.3962,E1 25.0895,E2 394.2654} C_DIS
LIN {X 42.1741,Y 69.1229,Z 82,A 53.8203,B 24.8908,C -2.4118,E1 25.0812,E2 390.7404} C_DIS
LIN {X 37.9627,Y 71.5228,Z 82,A 56.9087,B 24.8914,C -2.406,E1 25.0737,E2 387.6747} C_DIS
LIN {X 35.185,Y 72.929,Z 82,A 59.0456,B 24.8913,C -2.4067,E1 25.0684,E2 385.5418} C_DIS
LIN {X 31.723,Y 74.5007,Z 82,A 61.7499,B 24.891,C -2.4101,E1 25.0615,E2 382.8361} C_DIS
LIN {X 29.0723,Y 75.575,Z 82,A 63.791,B 24.8908,C -2.4126,E1 25.0562,E2 380.7936} C_DIS
LIN {X 26.1369,Y 76.6391,Z 82,A 66.3866,B 24.8895,C -2.4262,E1 25.0492,E2 378.171} C_DIS
LIN {X 22.6121,Y 77.7528,Z 82,A 69.0792,B 24.8892,C -2.4303,E1 25.042,E2 375.4733} C_DIS
LIN {X 19.1645,Y 78.6723,Z 82,A 71.1644,B 24.8902,C -2.4187,E1 25.0365,E2 373.4188} C_DIS
LIN {X 15.6638,Y 79.4442,Z 82,A 73.7024,B 24.8902,C -2.4199,E1 25.0295,E2 370.8812} C_DIS
LIN {X 12.9175,Y 79.9371,Z 82,A 76.0859,B 24.8889,C -2.4326,E1 25.0229,E2 368.4698} C_DIS
LIN {X 8.0082,Y 80.577,Z 82,A 79.2317,B 24.8898,C -2.4227,E1 25.0142,E2 365.3499} C_DIS
LIN {X 4.5969,Y 80.8424,Z 82,A 81.5283,B 24.8902,C -2.4191,E1 25.0079,E2 363.0627} C_DIS
LIN {X -0.2455,Y 80.9729,Z 82,A 84.9299,B 24.8902,C -2.4179,E1 24.9984,E2 359.6646} C_DIS
LIN {X -6.069,Y 80.746,Z 82,A 89.6799,B 24.8888,C -2.4344,E1 24.985,E2 354.8741} C_DIS
LIN {X -9.2657,Y 80.4412,Z 82,A 91.8614,B 24.8891,C -2.4305,E1 24.979,E2 352.7003} C_DIS
LIN {X -15.1805,Y 79.5373,Z 82,A 96.1061,B 24.8894,C -2.4277,E1 24.9673,E2 348.4582} C_DIS
LIN {X -18.8933,Y 78.7385,Z 82,A 99.0861,B 24.8889,C -2.4335,E1 24.9592,E2 345.4604} C_DIS
LIN {X -22.6268,Y 77.7484,Z 82,A 101.2392,B 24.8906,C -2.4142,E1 24.9535,E2 343.3496} C_DIS
LIN {X -25.9991,Y 76.6856,Z 82,A 103.47,B 24.8916,C -2.4038,E1 24.9476,E2 341.1397} C_DIS
LIN {X -29.1772,Y 75.5336,Z 82,A 106.2396,B 24.8909,C -2.4111,E1 24.9403,E2 338.3469} C_DIS
LIN {X -34.7957,Y 73.1161,Z 82,A 110.0309,B 24.8928,C -2.39,E1 24.9308,E2 334.5968} C_DIS
LIN {X -36.2973,Y 72.3819,Z 82,A 112.3135,B 24.8902,C -2.4183,E1 24.9249,E2 332.2406} C_DIS
LIN {X -39.8547,Y 70.4869,Z 82,A 114.6419,B 24.892,C -2.399,E1 24.9193,E2 329.9515} C_DIS
LIN {X -43.306,Y 68.421,Z 82,A 117.2939,B 24.8929,C -2.3884,E1 24.913,E2 327.3164} C_DIS
LIN {X -48.1708,Y 65.0873,Z 82,A 121.2562,B 24.8942,C -2.3744,E1 24.904,E2 323.3738} C_DIS
LIN {X -49.6794,Y 63.9421,Z 82,A 123.2221,B 24.8929,C -2.3885,E1 24.8996,E2 321.3673} C_DIS
LIN {X -53.415,Y 60.8563,Z 82,A 127.3561,B 24.8919,C -2.4,E1 24.8908,E2 317.1897} C_DIS
LIN {X -57.0695,Y 57.4434,Z 82,A 130.6132,B 24.8934,C -2.3839,E1 24.8844,E2 313.9571} C_DIS
LIN {X -59.9145,Y 54.4702,Z 82,A 132.6335,B 24.8961,C -2.3529,E1 24.8807,E2 312.0021} C_DIS
LIN {X -63.4798,Y 50.2686,Z 82,A 136.4822,B 24.8971,C -2.3415,E1 24.8738,E2 308.1627} C_DIS
LIN {X -65.2424,Y 47.959,Z 82,A 138.7645,B 24.8971,C -2.342,E1 24.87,E2 305.8684} C_DIS
LIN {X -67.3542,Y 44.947,Z 82,A 141.3691,B 24.8977,C -2.3349,E1 24.8659,E2 303.2678} C_DIS
LIN {X -70.0856,Y 40.5546,Z 82,A 145.1617,B 24.8983,C -2.328,E1 24.8604,E2 299.472} C_DIS
LIN {X -72.5779,Y 35.9035,Z 82,A 148.3257,B 24.9005,C -2.3023,E1 24.8563,E2 296.3526} C_DIS
LIN {X -73.3794,Y 34.2356,Z 82,A 150.0151,B 24.9,C -2.3083,E1 24.8543,E2 294.6399} C_DIS
LIN {X -74.6966,Y 31.2581,Z 82,A 152.2681,B 24.9007,C -2.3,E1 24.8518,E2 292.3941} C_DIS
LIN {X -75.917,Y 28.1678,Z 82,A 154.534,B 24.9016,C -2.2907,E1 24.8495,E2 290.1378} C_DIS
LIN {X -77.0219,Y 24.9848,Z 82,A 157.2119,B 24.9016,C -2.291,E1 24.8471,E2 287.444} C_DIS
LIN {X -78.1093,Y 21.3449,Z 82,A 159.9329,B 24.9022,C -2.2834,E1 24.845,E2 284.7252} C_DIS
LIN {X -78.8997,Y 18.2056,Z 82,A 162.428,B 24.9023,C -2.2816,E1 24.8434,E2 282.2199} C_DIS
LIN {X -79.8559,Y 13.4034,Z 82,A 165.4861,B 24.9042,C -2.26,E1 24.8418,E2 279.1951} C_DIS
LIN {X -80.5444,Y 8.3199,Z 82,A 169.3773,B 24.9046,C -2.2552,E1 24.8405,E2 275.2922} C_DIS
LIN {X -80.8671,Y 4.1267,Z 82,A 172.3841,B 24.9053,C -2.2465,E1 24.8399,E2 272.288} C_DIS
LIN {X -80.972,Y 0.4066,Z 82,A 175.1762,B 24.9057,C -2.2422,E1 24.8398,E2 269.4893} C_DIS
LIN {X -80.9266,Y -2.7519,Z 82,A 177.5558,B 24.906,C -2.2389,E1 24.84,E2 267.1034} C_DIS
LIN {X -80.6359,Y -7.3804,Z 82,A -179.2494,B 24.907,C -2.2263,E1 24.8407,E2 263.9196} C_DIS
LIN {X -79.9954,Y -12.5447,Z 82,A -175.339,B 24.9075,C -2.2207,E1 24.8422,E2 259.999} C_DIS
LIN {X -78.903,Y -18.1914,Z 82,A -171.8054,B 24.9097,C -2.1942,E1 24.8442,E2 256.508} C_DIS
LIN {X -78.2491,Y -20.8273,Z 82,A -170.0559,B 24.9105,C -2.1839,E1 24.8454,E2 254.7729} C_DIS
LIN {X -77.7048,Y -22.7738,Z 82,A -168.2362,B 24.9101,C -2.1898,E1 24.8468,E2 252.9286} C_DIS
LIN {X -76.5639,Y -26.3583,Z 82,A -165.4983,B 24.9105,C -2.1839,E1 24.8492,E2 250.1891} C_DIS
LIN {X -75.2224,Y -29.9725,Z 82,A -162.3145,B 24.9102,C -2.1881,E1 24.8525,E2 246.9774} C_DIS
LIN {X -73.9696,Y -32.9428,Z 82,A -160.7639,B 24.9123,C -2.1623,E1 24.8541,E2 245.4799} C_DIS
LIN {X -72.1099,Y -36.8343,Z 82,A -157.5967,B 24.9127,C -2.1569,E1 24.858,E2 242.3084} C_DIS
LIN {X -70.3368,Y -40.1176,Z 82,A -154.8017,B 24.913,C -2.1539,E1 24.8618,E2 239.5059} C_DIS
LIN {X -68.4265,Y -43.2972,Z 82,A -152.4088,B 24.914,C -2.1409,E1 24.8653,E2 237.1317} C_DIS
LIN {X -66.6591,Y -45.9699,Z 82,A -149.5799,B 24.9133,C -2.1503,E1 24.8697,E2 234.2664} C_DIS
LIN {X -63.46,Y -50.2936,Z 82,A -146.3832,B 24.9153,C -2.1247,E1 24.8751,E2 231.1153} C_DIS
LIN {X -60.975,Y -53.2791,Z 82,A -142.7432,B 24.9139,C -2.1426,E1 24.8818,E2 227.4161} C_DIS
LIN {X -58.6791,Y -55.7994,Z 82,A -140.2041,B 24.914,C -2.1409,E1 24.8867,E2 224.8701} C_DIS
LIN {X -56.1072,Y -58.3832,Z 82,A -137.8222,B 24.9149,C -2.1301,E1 24.8914,E2 222.5039} C_DIS
LIN {X -52.56,Y -61.5959,Z 82,A -135.0386,B 24.9167,C -2.107,E1 24.8972,E2 219.7645} C_DIS
LIN {X -50.4576,Y -63.3303,Z 82,A -133.0224,B 24.9168,C -2.1059,E1 24.9015,E2 217.7434} C_DIS
LIN {X -48.2774,Y -65.0085,Z 82,A -130.8825,B 24.9167,C -2.1078,E1 24.9063,E2 215.5911} C_DIS
LIN {X -44.9783,Y -67.3332,Z 82,A -128.0163,B 24.917,C -2.1035,E1 24.9129,E2 212.7255} C_DIS
LIN {X -40.7101,Y -69.9962,Z 82,A -124.2481,B 24.917,C -2.1042,E1 24.922,E2 208.9441} C_DIS
LIN {X -37.0717,Y -71.9886,Z 82,A -121.9926,B 24.9188,C -2.0812,E1 24.9274,E2 206.7369} C_DIS
LIN {X -34.5415,Y -73.237,Z 82,A -119.642,B 24.9182,C -2.0888,E1 24.9334,E2 204.3622} C_DIS
LIN {X -31.9726,Y -74.3945,Z 82,A -117.4899,B 24.918,C -2.0912,E1 24.9389,E2 202.1993} C_DIS
LIN {X -28.737,Y -75.7021,Z 82,A -114.816,B 24.9177,C -2.0947,E1 24.9459,E2 199.5113} C_DIS
LIN {X -25.4769,Y -76.8616,Z 82,A -112.239,B 24.9176,C -2.0965,E1 24.9528,E2 196.9254} C_DIS
LIN {X -21.2575,Y -78.1326,Z 82,A -109.3645,B 24.9183,C -2.0874,E1 24.9604,E2 194.0678} C_DIS
LIN {X -17.6409,Y -79.0289,Z 82,A -106.9725,B 24.9189,C -2.0789,E1 24.9669,E2 191.6927} C_DIS
LIN {X -13.4049,Y -79.8556,Z 82,A -103.6613,B 24.9184,C -2.0854,E1 24.976,E2 188.3627} C_DIS
LIN {X -9.527,Y -80.4106,Z 82,A -101.1339,B 24.919,C -2.0777,E1 24.983,E2 185.8518} C_DIS
LIN {X -5.863,Y -80.7614,Z 82,A -98.2028,B 24.9183,C -2.0873,E1 24.9912,E2 182.8967} C_DIS
LIN {X -1.1503,Y -80.9654,Z 82,A -95.0958,B 24.9188,C -2.0808,E1 24.9998,E2 179.8044} C_DIS
LIN {X -1.1503,Y -80.9654,Z 82,A -95.0958,B 24.9188,C -2.0808,E1 24.9998,E2 179.8044} C_DIS
Enddeposition()
LIN {X 0.5409,Y -79.9786,Z 82,A -94.6023,B 24.9191,C -2.0776,E1 25.0012,E2 179.3187} C_DIS
Startdeposition()
$VEL.CP = VEL_PRINT
LIN {X -2.5223,Y -79.9643,Z 82,A -98.0149,B 24.9218,C -2.0419,E1 24.9915,E2 182.8164} C_DIS
LIN {X -6.3465,Y -79.7519,Z 82,A -99.9537,B 24.9201,C -2.0647,E1 24.9862,E2 184.7017} C_DIS
LIN {X -9.1453,Y -79.4798,Z 82,A -102.177,B 24.9205,C -2.059,E1 24.98,E2 186.9401} C_DIS
LIN {X -12.477,Y -79.0255,Z 82,A -105.2118,B 24.9218,C -2.042,E1 24.9715,E2 190.0177} C_DIS
LIN {X -16.3296,Y -78.3202,Z 82,A -107.061,B 24.9197,C -2.0699,E1 24.9666,E2 191.8029} C_DIS
LIN {X -18.4555,Y -77.8476,Z 82,A -109.5221,B 24.9215,C -2.0455,E1 24.9598,E2 194.3252} C_DIS
LIN {X -22.0376,Y -76.9093,Z 82,A -111.3327,B 24.9196,C -2.0705,E1 24.955,E2 196.0791} C_DIS
LIN {X -25.044,Y -75.9844,Z 82,A -113.4815,B 24.9193,C -2.0751,E1 24.9493,E2 198.221} C_DIS
LIN {X -29.1118,Y -74.5196,Z 82,A -116.8014,B 24.9195,C -2.0716,E1 24.9406,E2 201.5558} C_DIS
LIN {X -32.1243,Y -73.2714,Z 82,A -119.1737,B 24.9195,C -2.073,E1 24.9345,E2 203.9303} C_DIS
LIN {X -36.6158,Y -71.1336,Z 82,A -122.0752,B 24.9177,C -2.0954,E1 24.9273,E2 206.7861} C_DIS
LIN {X -39.663,Y -69.4805,Z 82,A -124.8354,B 24.918,C -2.091,E1 24.9205,E2 209.5645} C_DIS
LIN {X -43.6033,Y -67.0792,Z 82,A -128.5532,B 24.9185,C -2.0847,E1 24.9116,E2 213.309} C_DIS
LIN {X -46.0934,Y -65.3931,Z 82,A -130.7196,B 24.9183,C -2.0878,E1 24.9066,E2 215.4753} C_DIS
LIN {X -48.5694,Y -63.5749,Z 82,A -132.9227,B 24.918,C -2.0916,E1 24.9017,E2 217.6774} C_DIS
LIN {X -51.6133,Y -61.1297,Z 82,A -135.6024,B 24.9173,C -2.0998,E1 24.8959,E2 220.3475} C_DIS
LIN {X -53.5901,Y -59.404,Z 82,A -137.9425,B 24.918,C -2.0913,E1 24.891,E2 222.7172} C_DIS
LIN {X -57.4182,Y -55.7123,Z 82,A -141.4023,B 24.9166,C -2.1084,E1 24.8842,E2 226.1508} C_DIS
LIN {X -60.247,Y -52.6398,Z 82,A -144.7685,B 24.9169,C -2.1053,E1 24.8778,E2 229.5394} C_DIS
LIN {X -62.9447,Y -49.3831,Z 82,A -148.2716,B 24.9173,C -2.1002,E1 24.8717,E2 233.0711} C_DIS
LIN {X -65.3044,Y -46.2176,Z 82,A -151.0712,B 24.9167,C -2.1079,E1 24.8672,E2 235.8661} C_DIS
LIN {X -67.4246,Y -43.0651,Z 82,A -152.9199,B 24.9143,C -2.1372,E1 24.8645,E2 237.6543} C_DIS
LIN {X -69.0024,Y -40.4893,Z 82,A -155.8154,B 24.9154,C -2.1241,E1 24.8603,E2 240.5959} C_DIS
LIN {X -70.6286,Y -37.5814,Z 82,A -157.6452,B 24.9137,C -2.1447,E1 24.8579,E2 242.3862} C_DIS
LIN {X -72.5196,Y -33.7869,Z 82,A -160.5044,B 24.9127,C -2.1576,E1 24.8544,E2 245.2301} C_DIS
LIN {X -73.4102,Y -31.8059,Z 82,A -162.7096,B 24.9137,C -2.1455,E1 24.8519,E2 247.4763} C_DIS
LIN {X -75.1589,Y -27.4186,Z 82,A -165.5532,B 24.9118,C -2.169,E1 24.8491,E2 250.28} C_DIS
LIN {X -75.9311,Y -25.2043,Z 82,A -167.7434,B 24.9124,C -2.161,E1 24.8471,E2 252.5017} C_DIS
LIN {X -77.306,Y -20.6032,Z 82,A -170.6289,B 24.9104,C -2.1853,E1 24.845,E2 255.346} C_DIS
LIN {X -77.9537,Y -17.9962,Z 82,A -173.8141,B 24.9125,C -2.1597,E1 24.8429,E2 258.6109} C_DIS
LIN {X -78.8836,Y -13.3432,Z 82,A -176.1618,B 24.9095,C -2.1963,E1 24.8418,E2 260.8851} C_DIS
LIN {X -79.465,Y -9.2687,Z 82,A -179.1591,B 24.9089,C -2.2043,E1 24.8407,E2 263.8813} C_DIS
LIN {X -79.7969,Y -5.7445,Z 82,A 177.9716,B 24.9089,C -2.2039,E1 24.84,E2 266.7686} C_DIS
LIN {X -79.9853,Y -1.7524,Z 82,A 175.1289,B 24.9081,C -2.2135,E1 24.8398,E2 269.6057} C_DIS
LIN {X -79.966,Y 2.4659,Z 82,A 172.3763,B 24.9067,C -2.2298,E1 24.8399,E2 272.3359} C_DIS
LIN {X -79.7677,Y 6.1489,Z 82,A 170.0788,B 24.9053,C -2.2468,E1 24.8403,E2 274.6066} C_DIS
LIN {X -79.4521,Y 9.3815,Z 82,A 167.1592,B 24.9059,C -2.2394,E1 24.8412,E2 277.5613} C_DIS
LIN {X -78.8416,Y 13.5927,Z 82,A 164.1734,B 24.905,C -2.2506,E1 24.8425,E2 280.5382} C_DIS
LIN {X -78.0603,Y 17.5303,Z 82,A 161.5668,B 24.9036,C -2.2664,E1 24.8439,E2 283.1225} C_DIS
LIN {X -77.5117,Y 19.8138,Z 82,A 159.2465,B 24.9045,C -2.2557,E1 24.8456,E2 285.4817} C_DIS
LIN {X -76.4958,Y 23.4332,Z 82,A 156.1098,B 24.9048,C -2.2531,E1 24.8481,E2 288.6427} C_DIS
LIN {X -75.1499,Y 27.4432,Z 82,A 154.0695,B 24.9019,C -2.2869,E1 24.85,E2 290.6138} C_DIS
LIN {X -73.9031,Y 30.6463,Z 82,A 151.3764,B 24.9017,C -2.2886,E1 24.8528,E2 293.3181} C_DIS
LIN {X -71.999,Y 34.8835,Z 82,A 148.3065,B 24.9003,C -2.3049,E1 24.8563,E2 296.3657} C_DIS
LIN {X -69.5219,Y 39.591,Z 82,A 144.2196,B 24.9,C -2.309,E1 24.8618,E2 300.4646} C_DIS
LIN {X -67.0519,Y 43.6453,Z 82,A 140.8105,B 24.8992,C -2.3183,E1 24.8668,E2 303.8689} C_DIS
LIN {X -65.6293,Y 45.7543,Z 82,A 138.355,B 24.9001,C -2.3073,E1 24.8708,E2 306.3626} C_DIS
LIN {X -63.4891,Y 48.6807,Z 82,A 136.1843,B 24.8986,C -2.3249,E1 24.8744,E2 308.5017} C_DIS
LIN {X -60.3831,Y 52.4839,Z 82,A 132.9584,B 24.8971,C -2.3413,E1 24.8801,E2 311.7033} C_DIS
LIN {X -57.4917,Y 55.6358,Z 82,A 129.839,B 24.8966,C -2.3474,E1 24.8861,E2 314.8217} C_DIS
LIN {X -55.3411,Y 57.776,Z 82,A 126.868,B 24.8979,C -2.3322,E1 24.8921,E2 317.8415} C_DIS
LIN {X -52.5163,Y 60.3548,Z 82,A 125.032,B 24.8954,C -2.3615,E1 24.8958,E2 319.6149} C_DIS
LIN {X -49.9531,Y 62.4932,Z 82,A 122.3546,B 24.8956,C -2.3592,E1 24.9017,E2 322.3078} C_DIS
LIN {X -46.0965,Y 65.3892,Z 82,A 118.5955,B 24.8956,C -2.3584,E1 24.9102,E2 326.0821} C_DIS
LIN {X -42.3657,Y 67.866,Z 82,A 115.1462,B 24.8956,C -2.3581,E1 24.9183,E2 329.5431} C_DIS
LIN {X -39.3484,Y 69.6599,Z 82,A 113.5268,B 24.8932,C -2.3859,E1 24.9221,E2 331.101} C_DIS
LIN {X -35.6648,Y 71.6149,Z 82,A 110.6927,B 24.8924,C -2.3949,E1 24.9291,E2 333.9215} C_DIS
LIN {X -33.0312,Y 72.8671,Z 82,A 107.9717,B 24.8936,C -2.3813,E1 24.936,E2 336.6819} C_DIS
LIN {X -29.8451,Y 74.2294,Z 82,A 105.1999,B 24.894,C -2.377,E1 24.9433,E2 339.4701} C_DIS
LIN {X -25.4581,Y 75.8455,Z 82,A 102.4818,B 24.8921,C -2.398,E1 24.9503,E2 342.1435} C_DIS
LIN {X -22.3939,Y 76.8069,Z 82,A 99.7878,B 24.8928,C -2.3899,E1 24.9575,E2 344.8613} C_DIS
LIN {X -18.2343,Y 77.8987,Z 82,A 97.0938,B 24.8916,C -2.4034,E1 24.9648,E2 347.5271} C_DIS
LIN {X -12.3012,Y 79.0527,Z 82,A 92.7875,B 24.8912,C -2.4073,E1 24.9766,E2 351.8286} C_DIS
LIN {X -6.9291,Y 79.7045,Z 82,A 88.8589,B 24.8912,C -2.408,E1 24.9875,E2 355.7582} C_DIS
LIN {X -1.1651,Y 79.9961,Z 82,A 84.5524,B 24.8915,C -2.4045,E1 24.9995,E2 360.0739} C_DIS
LIN {X 3.755,Y 79.9165,Z 82,A 81.2864,B 24.8908,C -2.4122,E1 25.0086,E2 363.3211} C_DIS
LIN {X 8.3429,Y 79.5678,Z 82,A 78.1374,B 24.8904,C -2.4161,E1 25.0173,E2 366.4592} C_DIS
LIN {X 13.4143,Y 78.8717,Z 82,A 74.3145,B 24.8909,C -2.4107,E1 25.0279,E2 370.2916} C_DIS
LIN {X 19.015,Y 77.7115,Z 82,A 70.1043,B 24.8914,C -2.4054,E1 25.0394,E2 374.5088} C_DIS
LIN {X 22.6711,Y 76.7246,Z 82,A 66.6063,B 24.8936,C -2.381,E1 25.049,E2 378.0589} C_DIS
LIN {X 26.1379,Y 75.6148,Z 82,A 64.6378,B 24.8922,C -2.3972,E1 25.054,E2 379.985} C_DIS
LIN {X 29.2752,Y 74.4554,Z 82,A 62.2658,B 24.8923,C -2.3956,E1 25.0602,E2 382.3557} C_DIS
LIN {X 33.6333,Y 72.5911,Z 82,A 59.0458,B 24.8922,C -2.397,E1 25.0684,E2 385.5646} C_DIS
LIN {X 37.2688,Y 70.7932,Z 82,A 55.8574,B 24.8933,C -2.385,E1 25.0764,E2 388.7728} C_DIS
LIN {X 40.2708,Y 69.1307,Z 82,A 53.3899,B 24.8936,C -2.3812,E1 25.0824,E2 391.2418} C_DIS
LIN {X 44.1658,Y 66.7087,Z 82,A 50.2982,B 24.8936,C -2.3819,E1 25.0897,E2 394.3219} C_DIS
LIN {X 46.446,Y 65.1415,Z 82,A 48.4085,B 24.8936,C -2.3814,E1 25.094,E2 396.2063} C_DIS
LIN {X 48.8463,Y 63.3615,Z 82,A 46.1314,B 24.8943,C -2.3735,E1 25.0991,E2 398.4939} C_DIS
LIN {X 50.9187,Y 61.7091,Z 82,A 43.3307,B 24.897,C -2.3429,E1 25.1052,E2 401.3562} C_DIS
LIN {X 54.2612,Y 58.7913,Z 82,A 40.8833,B 24.8956,C -2.3585,E1 25.1102,E2 403.7569} C_DIS
LIN {X 56.586,Y 56.5588,Z 82,A 38.6253,B 24.8959,C -2.3551,E1 25.1147,E2 406.0134} C_DIS
LIN {X 60.8284,Y 51.9669,Z 82,A 34.8241,B 24.895,C -2.3659,E1 25.1218,E2 409.7722} C_DIS
LIN {X 62.0082,Y 50.5537,Z 82,A 32.9118,B 24.8969,C -2.3446,E1 25.1252,E2 411.7262} C_DIS
LIN {X 64.3859,Y 47.4887,Z 82,A 29.9864,B 24.8978,C -2.3333,E1 25.1301,E2 414.6642} C_DIS
LIN {X 66.7667,Y 44.0779,Z 82,A 27.4524,B 24.8973,C -2.3396,E1 25.1341,E2 417.171} C_DIS
LIN {X 68.8861,Y 40.686,Z 82,A 24.4753,B 24.8983,C -2.3286,E1 25.1385,E2 420.1588} C_DIS
LIN {X 69.983,Y 38.7697,Z 82,A 22.7927,B 24.8989,C -2.3212,E1 25.1408,E2 421.8501} C_DIS
LIN {X 72.2481,Y 34.365,Z 82,A 19.0541,B 24.9003,C -2.3055,E1 25.1454,E2 425.606} C_DIS
LIN {X 73.8026,Y 30.8845,Z 82,A 16.8074,B 24.8996,C -2.3128,E1 25.1479,E2 427.823} C_DIS
LIN {X 74.9819,Y 27.9029,Z 82,A 14.2383,B 24.901,C -2.2976,E1 25.1505,E2 430.4138} C_DIS
LIN {X 76.2161,Y 24.3278,Z 82,A 11.9445,B 24.9005,C -2.3026,E1 25.1525,E2 432.6827} C_DIS
LIN {X 77.583,Y 19.5364,Z 82,A 8.5106,B 24.9011,C -2.2961,E1 25.1551,E2 436.1123} C_DIS
LIN {X 78.5202,Y 15.3387,Z 82,A 5.1143,B 24.9028,C -2.2766,E1 25.1571,E2 439.5349} C_DIS
LIN {X 79.1359,Y 11.7631,Z 82,A 2.0459,B 24.9047,C -2.2537,E1 25.1585,E2 442.6394} C_DIS
LIN {X 79.7835,Y 5.9507,Z 82,A -1.7112,B 24.9047,C -2.2541,E1 25.1595,E2 446.3732} C_DIS
LIN {X 79.9627,Y 2.5742,Z 82,A -3.7973,B 24.9044,C -2.2571,E1 25.1597,E2 448.4399} C_DIS
LIN {X 79.9967,Y -1.1363,Z 82,A -7.42,B 24.9077,C -2.2181,E1 25.1597,E2 452.1332} C_DIS
LIN {X 79.8531,Y -4.9333,Z 82,A -9.4519,B 24.9066,C -2.2312,E1 25.1594,E2 454.1222} C_DIS
LIN {X 79.6614,Y -7.3969,Z 82,A -12.1507,B 24.9095,C -2.1963,E1 25.1586,E2 456.8874} C_DIS
LIN {X 79.1046,Y -11.9657,Z 82,A -14.0698,B 24.9068,C -2.2292,E1 25.1579,E2 458.7173} C_DIS
LIN {X 78.0742,Y -17.4712,Z 82,A -18.4377,B 24.9088,C -2.2051,E1 25.1556,E2 463.1166} C_DIS
LIN {X 77.4089,Y -20.2139,Z 82,A -20.7305,B 24.91,C -2.1902,E1 25.154,E2 465.4315} C_DIS
LIN {X 76.1243,Y -24.6118,Z 82,A -23.9277,B 24.9106,C -2.1826,E1 25.1514,E2 468.6283} C_DIS
LIN {X 75.1961,Y -27.3168,Z 82,A -26.0144,B 24.9113,C -2.1751,E1 25.1494,E2 470.7211} C_DIS
LIN {X 73.557,Y -31.4675,Z 82,A -29.0923,B 24.9117,C -2.1691,E1 25.1461,E2 473.7962} C_DIS
LIN {X 71.8936,Y -35.1024,Z 82,A -31.7862,B 24.912,C -2.1659,E1 25.1429,E2 476.4831} C_DIS
LIN {X 70.1052,Y -38.5483,Z 82,A -34.8442,B 24.9134,C -2.1491,E1 25.1388,E2 479.5647} C_DIS
LIN {X 68.203,Y -41.8215,Z 82,A -37.9675,B 24.915,C -2.1285,E1 25.1343,E2 482.7207} C_DIS
LIN {X 66.054,Y -45.1401,Z 82,A -39.719,B 24.9129,C -2.1544,E1 25.1317,E2 484.4022} C_DIS
LIN {X 63.4138,Y -48.7785,Z 82,A -42.882,B 24.9135,C -2.1475,E1 25.1265,E2 487.5665} C_DIS
LIN {X 61.5043,Y -51.1651,Z 82,A -46.027,B 24.9163,C -2.112,E1 25.1207,E2 490.7808} C_DIS
LIN {X 59.1629,Y -53.8563,Z 82,A -48.3881,B 24.9163,C -2.1115,E1 25.1163,E2 493.1326} C_DIS
LIN {X 55.3776,Y -57.7408,Z 82,A -52.0669,B 24.9166,C -2.1085,E1 25.109,E2 496.8029} C_DIS
LIN {X 52.2785,Y -60.5625,Z 82,A -54.6652,B 24.9162,C -2.1141,E1 25.1037,E2 499.3776} C_DIS
LIN {X 48.5409,Y -63.5969,Z 82,A -58.194,B 24.917,C -2.1041,E1 25.096,E2 502.9168} C_DIS
LIN {X 46.168,Y -65.3398,Z 82,A -61.0524,B 24.9191,C -2.077,E1 25.0893,E2 505.8295} C_DIS
LIN {X 42.9882,Y -67.474,Z 82,A -62.8488,B 24.9173,C -2.1005,E1 25.0853,E2 507.5645} C_DIS
LIN {X 39.073,Y -69.8137,Z 82,A -66.1701,B 24.9179,C -2.0929,E1 25.0773,E2 510.8935} C_DIS
LIN {X 35.2212,Y -71.8339,Z 82,A -69.7151,B 24.9193,C -2.0747,E1 25.0683,E2 514.4718} C_DIS
LIN {X 31.3569,Y -73.6036,Z 82,A -72.1353,B 24.9182,C -2.0889,E1 25.0623,E2 516.8525} C_DIS
LIN {X 28.6024,Y -74.717,Z 82,A -74.6814,B 24.9194,C -2.0734,E1 25.0556,E2 519.4296} C_DIS
LIN {X 24.2451,Y -76.2429,Z 82,A -77.6085,B 24.9188,C -2.0806,E1 25.0479,E2 522.3339} C_DIS
LIN {X 21.7485,Y -76.9912,Z 82,A -79.9352,B 24.92,C -2.0649,E1 25.0416,E2 524.6939} C_DIS
LIN {X 15.5398,Y -78.4814,Z 82,A -84.0165,B 24.9192,C -2.0751,E1 25.0306,E2 528.7453} C_DIS
LIN {X 12.1188,Y -79.0809,Z 82,A -87.2974,B 24.9212,C -2.0501,E1 25.0214,E2 532.0824} C_DIS
LIN {X 8.8679,Y -79.5123,Z 82,A -90.5029,B 24.9232,C -2.0242,E1 25.0123,E2 535.3471} C_DIS
LIN {X 3.1133,Y -79.9441,Z 82,A -92.9813,B 24.9196,C -2.07,E1 25.0057,E2 537.716} C_DIS
LIN {X 0.5409,Y -79.9786,Z 82,A -94.5994,B 24.9192,C -2.0763,E1 25.0012,E2 539.3187} C_DIS
Enddeposition()
LIN {X 0.5409,Y -79.9786,Z 82,A -94.5994,B 24.9192,C -2.0763,E1 25.0012,E2 539.3187} C_DIS
Startdeposition()
$VEL.CP = VEL_PRINT
LIN {X 2.8522,Y -78.9848,Z 82,A -92.4914,B 24.9168,C -2.1058,E1 25.0073,E2 537.1413} C_DIS
LIN {X 9.2565,Y -78.4913,Z 82,A -87.2747,B 24.9153,C -2.1246,E1 25.0219,E2 531.883} C_DIS
LIN {X 14.6608,Y -77.664,Z 82,A -83.7424,B 24.9161,C -2.1148,E1 25.0316,E2 528.3776} C_DIS
LIN {X 19.32,Y -76.6383,Z 82,A -80.1657,B 24.9156,C -2.1215,E1 25.0413,E2 524.7899} C_DIS
LIN {X 23.3183,Y -75.517,Z 82,A -77.4721,B 24.9161,C -2.1154,E1 25.0485,E2 522.1154} C_DIS
LIN {X 28.4523,Y -73.7377,Z 82,A -73.1904,B 24.9149,C -2.1307,E1 25.0598,E2 517.8061} C_DIS
LIN {X 32.467,Y -72.0587,Z 82,A -69.7492,B 24.9138,C -2.1442,E1 25.0687,E2 514.3414} C_DIS
LIN {X 37.29,Y -69.6866,Z 82,A -66.456,B 24.9147,C -2.1321,E1 25.0768,E2 511.0858} C_DIS
LIN {X 39.327,Y -68.5562,Z 82,A -64.348,B 24.9135,C -2.148,E1 25.082,E2 508.9465} C_DIS
LIN {X 42.2458,Y -66.7985,Z 82,A -61.8477,B 24.913,C -2.1536,E1 25.0879,E2 506.441} C_DIS
LIN {X 46.4954,Y -63.9124,Z 82,A -57.2147,B 24.9101,C -2.1896,E1 25.0986,E2 501.739} C_DIS
LIN {X 50.7076,Y -60.6248,Z 82,A -54.5755,B 24.9125,C -2.1594,E1 25.1041,E2 499.1814} C_DIS
LIN {X 53.8915,Y -57.8133,Z 82,A -51.709,B 24.9125,C -2.1598,E1 25.11,E2 496.3253} C_DIS
LIN {X 55.4788,Y -56.291,Z 82,A -49.0253,B 24.9094,C -2.1979,E1 25.1155,E2 493.5629} C_DIS
LIN {X 58.5648,Y -53.075,Z 82,A -45.5765,B 24.9081,C -2.2129,E1 25.122,E2 490.0938} C_DIS
LIN {X 61.8476,Y -49.2087,Z 82,A -43.4675,B 24.9114,C -2.1729,E1 25.1255,E2 488.0892} C_DIS
LIN {X 65.0628,Y -44.8718,Z 82,A -39.9111,B 24.9114,C -2.1722,E1 25.1314,E2 484.5515} C_DIS
LIN {X 66.931,Y -42.0336,Z 82,A -36.9142,B 24.9096,C -2.1958,E1 25.1361,E2 481.5138} C_DIS
LIN {X 68.07,Y -40.1626,Z 82,A -34.885,B 24.908,C -2.2143,E1 25.139,E2 479.4513} C_DIS
LIN {X 70.6564,Y -35.4168,Z 82,A -30.8804,B 24.9068,C -2.2285,E1 25.1442,E2 475.4344} C_DIS
LIN {X 72.6002,Y -31.2396,Z 82,A -27.8155,B 24.9068,C -2.2297,E1 25.1477,E2 472.3833} C_DIS
LIN {X 74.2426,Y -27.1033,Z 82,A -25.1217,B 24.9073,C -2.2226,E1 25.1503,E2 469.7211} C_DIS
LIN {X 75.2731,Y -24.0945,Z 82,A -22.3724,B 24.9055,C -2.2439,E1 25.1528,E2 466.9373} C_DIS
LIN {X 76.782,Y -18.737,Z 82,A -18.8316,B 24.9058,C -2.2407,E1 25.1554,E2 463.4242} C_DIS
LIN {X 77.8034,Y -13.8983,Z 82,A -14.8779,B 24.9039,C -2.2638,E1 25.1576,E2 459.439} C_DIS
LIN {X 78.4958,Y -9.2181,Z 82,A -10.9907,B 24.9017,C -2.2894,E1 25.159,E2 455.5144} C_DIS
LIN {X 78.9619,Y -3.4012,Z 82,A -7.1019,B 24.9014,C -2.2919,E1 25.1597,E2 451.6427} C_DIS
LIN {X 79.0337,Y 0.4208,Z 82,A -4.2442,B 24.9004,C -2.3035,E1 25.1597,E2 448.7747} C_DIS
LIN {X 78.898,Y 4.6646,Z 82,A -1.2531,B 24.8998,C -2.3105,E1 25.1593,E2 445.7849} C_DIS
LIN {X 78.5555,Y 8.7077,Z 82,A 1.5411,B 24.8994,C -2.315,E1 25.1586,E2 442.9965} C_DIS
LIN {X 78.0111,Y 12.6864,Z 82,A 4.3146,B 24.899,C -2.3197,E1 25.1574,E2 440.2283} C_DIS
LIN {X 77.3213,Y 16.3702,Z 82,A 7.5489,B 24.8969,C -2.3446,E1 25.1556,E2 436.954} C_DIS
LIN {X 75.6509,Y 22.8839,Z 82,A 11.54,B 24.898,C -2.3312,E1 25.1528,E2 433.0175} C_DIS
LIN {X 74.4982,Y 26.3937,Z 82,A 14.6902,B 24.896,C -2.354,E1 25.1499,E2 429.8312} C_DIS
LIN {X 73.1924,Y 29.8233,Z 82,A 17.1072,B 24.896,C -2.354,E1 25.1475,E2 427.4276} C_DIS
LIN {X 71.3105,Y 34.0792,Z 82,A 20.4585,B 24.8952,C -2.3628,E1 25.1436,E2 424.0737} C_DIS
LIN {X 69.2725,Y 38.0533,Z 82,A 23.4567,B 24.8952,C -2.3641,E1 25.1397,E2 421.0882} C_DIS
LIN {X 67.5302,Y 41.0637,Z 82,A 26.422,B 24.8933,C -2.3846,E1 25.1355,E2 418.0897} C_DIS
LIN {X 66.1326,Y 43.2795,Z 82,A 28.1784,B 24.8933,C -2.385,E1 25.1328,E2 416.3412} C_DIS
LIN {X 63.2413,Y 47.4036,Z 82,A 31.8142,B 24.8925,C -2.3935,E1 25.1269,E2 412.7029} C_DIS
LIN {X 60.5032,Y 50.8539,Z 82,A 34.8267,B 24.8923,C -2.3954,E1 25.1216,E2 409.6999} C_DIS
LIN {X 57.5875,Y 54.1317,Z 82,A 38.557,B 24.8901,C -2.4194,E1 25.1145,E2 405.9294} C_DIS
LIN {X 55.1906,Y 56.5755,Z 82,A 41.1731,B 24.8893,C -2.4287,E1 25.1093,E2 403.3022} C_DIS
LIN {X 52.7846,Y 58.8248,Z 82,A 43.3557,B 24.8894,C -2.4271,E1 25.1048,E2 401.1321} C_DIS
LIN {X 49.6674,Y 61.4794,Z 82,A 45.932,B 24.89,C -2.4207,E1 25.0993,E2 398.5807} C_DIS
LIN {X 46.9911,Y 63.5495,Z 82,A 48.6003,B 24.889,C -2.4316,E1 25.0933,E2 395.8965} C_DIS
LIN {X 43.7397,Y 65.8292,Z 82,A 51.4618,B 24.8887,C -2.4357,E1 25.0867,E2 393.0348} C_DIS
LIN {X 40.5982,Y 67.8108,Z 82,A 54.0193,B 24.8887,C -2.4357,E1 25.0806,E2 390.4854} C_DIS
LIN {X 36.8517,Y 69.9179,Z 82,A 56.5615,B 24.8898,C -2.4229,E1 25.0745,E2 387.981} C_DIS
LIN {X 33.3659,Y 71.6469,Z 82,A 59.4346,B 24.8894,C -2.4278,E1 25.0673,E2 385.1038} C_DIS
LIN {X 29.9176,Y 73.154,Z 82,A 62.0966,B 24.8893,C -2.4288,E1 25.0605,E2 382.4458} C_DIS
LIN {X 26.487,Y 74.4655,Z 82,A 66.3149,B 24.8848,C -2.477,E1 25.0491,E2 378.122} C_DIS
LIN {X 21.8547,Y 75.9541,Z 82,A 68.4044,B 24.8885,C -2.4375,E1 25.0438,E2 376.1301} C_DIS
LIN {X 18.5654,Y 76.8239,Z 82,A 72.2477,B 24.8847,C -2.4789,E1 25.0331,E2 372.194} C_DIS
LIN {X 13.9622,Y 77.7921,Z 82,A 74.5712,B 24.8875,C -2.4488,E1 25.027,E2 369.9448} C_DIS
LIN {X 8.6864,Y 78.5577,Z 82,A 78.2329,B 24.8879,C -2.4438,E1 25.0169,E2 366.2979} C_DIS
LIN {X 3.8635,Y 78.9421,Z 82,A 81.8657,B 24.8876,C -2.4475,E1 25.0067,E2 362.6582} C_DIS
LIN {X -0.9224,Y 79.031,Z 82,A 85.2823,B 24.8878,C -2.4454,E1 24.9972,E2 359.2469} C_DIS
LIN {X -5.5713,Y 78.8389,Z 82,A 88.5745,B 24.8881,C -2.4419,E1 24.9881,E2 355.962} C_DIS
LIN {X -7.9315,Y 78.6367,Z 82,A 90.8727,B 24.8867,C -2.4572,E1 24.9815,E2 353.6262} C_DIS
LIN {X -12.5865,Y 78.0278,Z 82,A 94.7746,B 24.8856,C -2.4688,E1 24.9707,E2 349.6934} C_DIS
LIN {X -16.5242,Y 77.2892,Z 82,A 96.5354,B 24.8887,C -2.4349,E1 24.9661,E2 348.0113} C_DIS
LIN {X -18.8375,Y 76.7575,Z 82,A 99.053,B 24.8869,C -2.4551,E1 24.9591,E2 345.4422} C_DIS
LIN {X -22.161,Y 75.8654,Z 82,A 101.47,B 24.8873,C -2.4503,E1 24.9527,E2 343.0327} C_DIS
LIN {X -26.7397,Y 74.3752,Z 82,A 105.4296,B 24.8865,C -2.4587,E1 24.9422,E2 339.0452} C_DIS
LIN {X -30.5243,Y 72.9031,Z 82,A 107.1881,B 24.8898,C -2.4227,E1 24.9378,E2 337.3686} C_DIS
LIN {X -34.9245,Y 70.9005,Z 82,A 110.9385,B 24.8898,C -2.4239,E1 24.9283,E2 333.6061} C_DIS
LIN {X -38.9248,Y 68.7868,Z 82,A 114.3761,B 24.8898,C -2.4225,E1 24.9198,E2 330.162} C_DIS
LIN {X -41.7646,Y 67.0991,Z 82,A 116.6479,B 24.8906,C -2.4149,E1 24.9144,E2 327.9013} C_DIS
LIN {X -43.9279,Y 65.7048,Z 82,A 118.9465,B 24.8898,C -2.4227,E1 24.909,E2 325.5765} C_DIS
LIN {X -47.7172,Y 63.0057,Z 82,A 121.9953,B 24.8912,C -2.4074,E1 24.9022,E2 322.5536} C_DIS
LIN {X -50.2313,Y 61.0205,Z 82,A 124.4723,B 24.8913,C -2.4064,E1 24.8968,E2 320.0697} C_DIS
LIN {X -53.669,Y 58.0193,Z 82,A 127.6281,B 24.8924,C -2.3949,E1 24.8903,E2 316.9286} C_DIS
LIN {X -55.739,Y 56.0339,Z 82,A 130.2445,B 24.8916,C -2.4039,E1 24.885,E2 314.2797} C_DIS
LIN {X -59.2113,Y 52.3527,Z 82,A 133.6694,B 24.8929,C -2.3885,E1 24.8786,E2 310.8765} C_DIS
LIN {X -61.7947,Y 49.2757,Z 82,A 136.3947,B 24.8941,C -2.3761,E1 24.8738,E2 308.168} C_DIS
LIN {X -64.1318,Y 46.1916,Z 82,A 139.5378,B 24.8939,C -2.3773,E1 24.8686,E2 305.0069} C_DIS
LIN {X -65.9007,Y 43.6312,Z 82,A 142.4706,B 24.8929,C -2.3885,E1 24.864,E2 302.0327} C_DIS
LIN {X -68.3058,Y 39.7628,Z 82,A 144.7073,B 24.8962,C -2.3518,E1 24.8609,E2 299.8721} C_DIS
LIN {X -70.4576,Y 35.8095,Z 82,A 147.7094,B 24.8976,C -2.3357,E1 24.857,E2 296.8924} C_DIS
LIN {X -71.4166,Y 33.8585,Z 82,A 150.0446,B 24.8964,C -2.3503,E1 24.8541,E2 294.5098} C_DIS
LIN {X -72.927,Y 30.4669,Z 82,A 152.2213,B 24.8982,C -2.3292,E1 24.8518,E2 292.3715} C_DIS
LIN {X -73.6606,Y 28.6487,Z 82,A 153.7986,B 24.8982,C -2.3288,E1 24.8501,E2 290.7863} C_DIS
LIN {X -75.2732,Y 24.0937,Z 82,A 157.344,B 24.8991,C -2.3191,E1 24.8469,E2 287.244} C_DIS
LIN {X -76.4584,Y 20.0193,Z 82,A 160.4502,B 24.8999,C -2.3102,E1 24.8446,E2 284.1408} C_DIS
LIN {X -77.2176,Y 16.8523,Z 82,A 162.7622,B 24.9006,C -2.3016,E1 24.8432,E2 281.8359} C_DIS
LIN {X -77.8244,Y 13.7825,Z 82,A 165.5269,B 24.9002,C -2.3069,E1 24.8418,E2 279.0421} C_DIS
LIN {X -78.3401,Y 10.4622,Z 82,A 168.2493,B 24.9002,C -2.3064,E1 24.8408,E2 276.3046} C_DIS
LIN {X -78.743,Y 6.8052,Z 82,A 170.0829,B 24.9027,C -2.2768,E1 24.8403,E2 274.5307} C_DIS
LIN {X -78.991,Y 2.6516,Z 82,A 173.9424,B 24.9017,C -2.2885,E1 24.8398,E2 270.62} C_DIS
LIN {X -79.0309,Y -0.9441,Z 82,A 175.9627,B 24.9037,C -2.2654,E1 24.8398,E2 268.6429} C_DIS
LIN {X -78.9297,Y -4.0902,Z 82,A 178.8316,B 24.9031,C -2.273,E1 24.8402,E2 265.7384} C_DIS
LIN {X -78.6763,Y -7.5282,Z 82,A -178.6936,B 24.9038,C -2.2645,E1 24.8409,E2 263.269} C_DIS
LIN {X -78.2896,Y -10.8345,Z 82,A -176.8391,B 24.9056,C -2.2428,E1 24.8416,E2 261.4554} C_DIS
LIN {X -77.753,Y -14.18,Z 82,A -173.6592,B 24.9047,C -2.2536,E1 24.8431,E2 258.2308} C_DIS
LIN {X -77.0044,Y -17.8011,Z 82,A -172.0142,B 24.9076,C -2.2191,E1 24.8441,E2 256.6586} C_DIS
LIN {X -76.509,Y -19.8232,Z 82,A -169.7713,B 24.9065,C -2.2331,E1 24.8457,E2 254.369} C_DIS
LIN {X -74.6613,Y -25.9289,Z 82,A -165.8774,B 24.9091,C -2.2008,E1 24.8489,E2 250.5301} C_DIS
LIN {X -73.9276,Y -27.9513,Z 82,A -163.7882,B 24.9084,C -2.2097,E1 24.8509,E2 248.4077} C_DIS
LIN {X -72.0072,Y -32.5812,Z 82,A -159.8679,B 24.9087,C -2.2068,E1 24.8553,E2 244.4727} C_DIS
LIN {X -70.4217,Y -35.8797,Z 82,A -157.7053,B 24.9103,C -2.1868,E1 24.858,E2 242.3462} C_DIS
LIN {X -67.7105,Y -40.7671,Z 82,A -153.5223,B 24.9109,C -2.1794,E1 24.8637,E2 238.159} C_DIS
LIN {X -65.478,Y -44.2628,Z 82,A -150.2499,B 24.9109,C -2.1787,E1 24.8688,E2 234.8719} C_DIS
LIN {X -62.2817,Y -48.6595,Z 82,A -146.7882,B 24.9128,C -2.1566,E1 24.8745,E2 231.4462} C_DIS
LIN {X -58.3092,Y -53.3536,Z 82,A -142.1371,B 24.9132,C -2.1515,E1 24.883,E2 226.7861} C_DIS
LIN {X -56.1953,Y -55.5756,Z 82,A -139.02,B 24.9116,C -2.1706,E1 24.8892,E2 223.6101} C_DIS
LIN {X -53.3297,Y -58.3312,Z 82,A -136.7436,B 24.9134,C -2.1486,E1 24.8938,E2 221.377} C_DIS
LIN {X -50.4687,Y -60.8232,Z 82,A -133.9911,B 24.9138,C -2.1435,E1 24.8996,E2 218.6261} C_DIS
LIN {X -47.4384,Y -63.2152,Z 82,A -131.5623,B 24.915,C -2.1286,E1 24.9049,E2 216.2238} C_DIS
LIN {X -45.2957,Y -64.7681,Z 82,A -129.4471,B 24.9149,C -2.1307,E1 24.9098,E2 214.0964} C_DIS
LIN {X -39.5129,Y -68.4494,Z 82,A -124.7569,B 24.9161,C -2.1156,E1 24.9208,E2 209.4272} C_DIS
LIN {X -36.2621,Y -70.2263,Z 82,A -121.81,B 24.9158,C -2.1192,E1 24.9281,E2 206.4634} C_DIS
LIN {X -32.7019,Y -71.9528,Z 82,A -119.2493,B 24.9167,C -2.1074,E1 24.9345,E2 203.9243} C_DIS
LIN {X -29.7266,Y -73.2318,Z 82,A -116.1221,B 24.9152,C -2.1266,E1 24.9427,E2 200.7444} C_DIS
LIN {X -24.7947,Y -75.0468,Z 82,A -112.9216,B 24.9168,C -2.1063,E1 24.951,E2 197.5857} C_DIS
LIN {X -21.5882,Y -76.0297,Z 82,A -109.075,B 24.9137,C -2.1448,E1 24.9616,E2 193.6415} C_DIS
LIN {X -16.6071,Y -77.2711,Z 82,A -106.8607,B 24.9173,C -2.1001,E1 24.9674,E2 191.5306} C_DIS
LIN {X -12.6324,Y -78.0194,Z 82,A -103.8217,B 24.9171,C -2.102,E1 24.9757,E2 188.4837} C_DIS
LIN {X -6.8954,Y -78.7347,Z 82,A -98.9772,B 24.9157,C -2.1202,E1 24.9893,E2 183.5931} C_DIS
LIN {X -1.8318,Y -79.0148,Z 82,A -94.6982,B 24.9142,C -2.1383,E1 25.0013,E2 179.2705} C_DIS
LIN {X -1.8318,Y -79.0148,Z 82,A -94.6982,B 24.9142,C -2.1383,E1 25.0013,E2 179.2705} C_DIS
Enddeposition()
LIN {X 0.5236,Y -78.0475,Z 82,A -94.3447,B 24.916,C -2.1162,E1 25.0022,E2 178.9694} C_DIS
Startdeposition()
$VEL.CP = VEL_PRINT
LIN {X -2.0869,Y -78.039,Z 82,A -97.5632,B 24.9189,C -2.079,E1 24.993,E2 182.2764} C_DIS
LIN {X -6.7241,Y -77.7775,Z 82,A -101.2845,B 24.9196,C -2.0705,E1 24.9825,E2 186.0196} C_DIS
LIN {X -10.5865,Y -77.3456,Z 82,A -103.1981,B 24.9176,C -2.0968,E1 24.9774,E2 187.8722} C_DIS
LIN {X -14.279,Y -76.7507,Z 82,A -106.1458,B 24.9179,C -2.092,E1 24.9692,E2 190.834} C_DIS
LIN {X -17.4435,Y -76.0926,Z 82,A -109.2731,B 24.9194,C -2.0727,E1 24.9606,E2 194.0111} C_DIS
LIN {X -21.2726,Y -75.1121,Z 82,A -111.5811,B 24.918,C -2.0905,E1 24.9545,E2 196.2805} C_DIS
LIN {X -25.1162,Y -73.9159,Z 82,A -114.4141,B 24.9176,C -2.096,E1 24.947,E2 199.1055} C_DIS
LIN {X -30.0117,Y -72.0677,Z 82,A -118.1832,B 24.9172,C -2.1016,E1 24.9372,E2 202.8695} C_DIS
LIN {X -33.2125,Y -70.6496,Z 82,A -120.9748,B 24.9174,C -2.0985,E1 24.9301,E2 205.6752} C_DIS
LIN {X -36.0539,Y -69.243,Z 82,A -123.384,B 24.9174,C -2.0993,E1 24.9241,E2 208.0893} C_DIS
LIN {X -38.7605,Y -67.7643,Z 82,A -125.2292,B 24.9162,C -2.1134,E1 24.9197,E2 209.9063} C_DIS
LIN {X -41.9456,Y -65.8398,Z 82,A -128.5344,B 24.9171,C -2.1025,E1 24.9117,E2 213.2478} C_DIS
LIN {X -45.7533,Y -63.255,Z 82,A -131.245,B 24.9153,C -2.1253,E1 24.9056,E2 215.9133} C_DIS
LIN {X -47.9706,Y -61.59,Z 82,A -133.6541,B 24.9158,C -2.1191,E1 24.9002,E2 218.3457} C_DIS
LIN {X -51.143,Y -58.9816,Z 82,A -136.8866,B 24.9158,C -2.1193,E1 24.8933,E2 221.5905} C_DIS
LIN {X -54.9637,Y -55.4379,Z 82,A -140.4049,B 24.9145,C -2.1348,E1 24.8862,E2 225.0862} C_DIS
LIN {X -56.6384,Y -53.7267,Z 82,A -142.4015,B 24.9147,C -2.1325,E1 24.8824,E2 227.0969} C_DIS
LIN {X -59.8136,Y -50.1678,Z 82,A -145.7303,B 24.9137,C -2.1448,E1 24.8763,E2 230.4115} C_DIS
LIN {X -61.595,Y -47.9642,Z 82,A -148.0316,B 24.9137,C -2.1441,E1 24.8723,E2 232.7253} C_DIS
LIN {X -64.2637,Y -44.3238,Z 82,A -151.433,B 24.9133,C -2.1501,E1 24.8668,E2 236.1291} C_DIS
LIN {X -66.2974,Y -41.2193,Z 82,A -153.7497,B 24.9119,C -2.1672,E1 24.8634,E2 238.4166} C_DIS
LIN {X -69.0188,Y -36.4796,Z 82,A -157.8224,B 24.9112,C -2.1764,E1 24.8578,E2 242.4888} C_DIS
LIN {X -70.0828,Y -34.3925,Z 82,A -159.8511,B 24.9114,C -2.1734,E1 24.8552,E2 244.5355} C_DIS
LIN {X -72.9522,Y -27.7912,Z 82,A -164.7951,B 24.9095,C -2.1968,E1 24.8499,E2 249.451} C_DIS
LIN {X -74.1937,Y -24.2838,Z 82,A -167.8549,B 24.9095,C -2.1968,E1 24.8471,E2 252.5283} C_DIS
LIN {X -75.7097,Y -19.041,Z 82,A -171.7065,B 24.9082,C -2.2126,E1 24.8443,E2 256.3646} C_DIS
LIN {X -76.6058,Y -15.0289,Z 82,A -174.8453,B 24.9076,C -2.2189,E1 24.8424,E2 259.5067} C_DIS
LIN {X -77.1951,Y -11.6341,Z 82,A -177.3282,B 24.9069,C -2.2279,E1 24.8413,E2 261.983} C_DIS
LIN {X -77.707,Y -7.4878,Z 82,A 179.2563,B 24.9068,C -2.229,E1 24.8403,E2 265.4162} C_DIS
LIN {X -78.0018,Y -3.1778,Z 82,A 176.4168,B 24.9053,C -2.2471,E1 24.8399,E2 268.2297} C_DIS
LIN {X -78.0673,Y 0.0507,Z 82,A 173.6271,B 24.9055,C -2.2445,E1 24.8399,E2 271.0425} C_DIS
Enddeposition()
END
